KUKA KRL program: EPS_2_251112_SAMH04_A_20250918010312.src

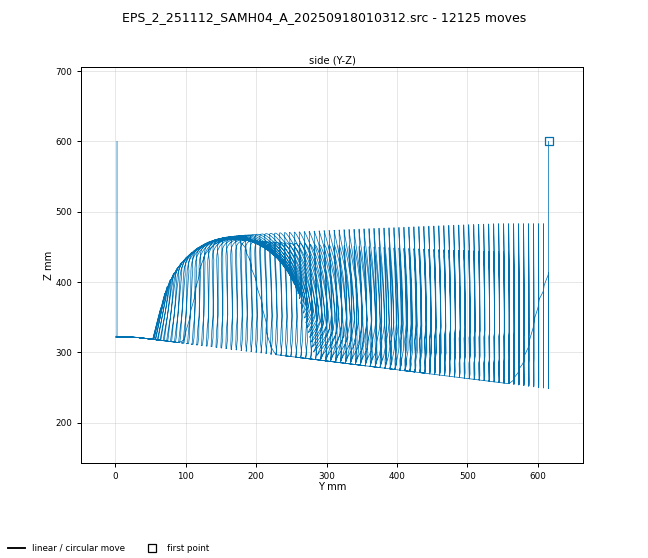
[picture p0: tool path of EPS_2_251112_SAMH04_A_20250918010312.src, 12125 of 12127 moves have a stored position in this frame; points joined in program order, loops and branches not executed]
&ACCESS RVP
&REL 4
&COMMENT QRS 19112012
&PARAM EDITMASK = *
DEF PART()
EXT BAS (BAS_COMMAND :IN,REAL :IN )
INT I
BAS (#INITMOV,0 )

;KUKA QRS Post kuka4.cps  Date:22-06-2017 !

File_ID=2832

QRS_PRE_INIT()

;Init var - Until changes are made in qrs_pre_init
Outlet_Square_prg=0
Inlet_1_Square_prg=0
Inlet_2_Square_prg=0
Inlet_3_Square_prg=0
Inlet_4_Square_prg=0
Inlet_5_Square_prg=0

Outlet_1={X 0.000, Y 541.230, Z 408.000, B 0.000, E1 0.000 }
Inlet_1={X 0.000, Y 544.070, Z 368.000, B 0.000, E1 90.000 }
Outlet_1_type=150
Inlet_1_type=150
;QRS#1=Sidecore dimensions
;QRS#2=150-6" PVC SDR 28
;QRS#3=150-6" PVC SDR 28
;QRS#4=
;QRS#5=
;QRS#6=
;QRS#7=
;QRS#8=
;QRS#9=10-06 PSX
;QRS#10=10-06 PSX
;QRS#11=
;QRS#12=
;QRS#13=
;QRS#14=
;QRS#15=
;QRS#16=1220x127x762 2,5'
;QRS#17=EPS Height
;QRS#18=483
;QRS#19=*
;QRS#20= UPDATED VERSION 22-06-2017
;QRS#21=*
Outlet_Square=070
Inlet_1_Square=070
Inlet_2_Square=0
Inlet_3_Square=0
Inlet_4_Square=0
Inlet_5_Square=0
Mill_Square=1
Outlet_Square_Prg=203
Inlet_1_Square_prg=203

QRS_INIT()

$ADVANCE=5

; T1
PTP {E1 173.474,E2 173.474}
PTP {X 0,Y 615.498,A -85,B 0,C 180,E1 173.474,E2 173.474,E3 0,E4 0,E5 0,E6 0}
QRS_SPEED_INIT()
LIN {X 0,Y 615.498,Z 600,A -85,B 0,C 180,E1 173.474,E2 173.474,E3 0,E4 0,E5 0,E6 0} C_VEL
LIN {X 0,Y 615.498,Z 427.975,A -85,B 0,C 180,E1 173.474,E2 173.474} C_VEL
LIN {X 0,Y 615.498,Z 415.28,A -85,B 0,C 180,E1 173.474,E2 173.474} C_VEL
LIN {X 0,Y 615.497,Z 413.833,A -85,B 0,C 180,E1 173.417,E2 173.417} C_VEL
LIN {X 0,Y 615.484,Z 405.601,A -85,B 0,C 180,E1 172.706,E2 172.706} C_VEL
LIN {X 0,Y 615.494,Z 395.743,A -85,B 0,C 180,E1 172.046,E2 172.046} C_VEL
LIN {X 0,Y 615.487,Z 388.006,A -85,B 0,C 180,E1 171.633,E2 171.633} C_VEL
LIN {X 0,Y 615.488,Z 379.171,A -85,B 0,C 180,E1 171.26,E2 171.26} C_VEL
LIN {X 0,Y 615.479,Z 369.995,A -85,B 0,C 180,E1 170.971,E2 170.971} C_VEL
LIN {X 0,Y 615.472,Z 360.409,A -85,B 0,C 180,E1 170.763,E2 170.763} C_VEL
LIN {X 0,Y 615.49,Z 301.527,A -85,B 0,C 180,E1 170.059,E2 170.059} C_VEL
LIN {X 0,Y 615.48,Z 284.33,A -85,B 0,C 180,E1 169.851,E2 169.851} C_VEL
LIN {X 0,Y 615.493,Z 270.832,A -85,B 0,C 180,E1 167.139,E2 167.139} C_VEL
LIN {X 0,Y 615.447,Z 257.533,A -85,B 0,C 180,E1 164.438,E2 164.438} C_VEL
LIN {X 0,Y 615.433,Z 248.511,A -85,B 0,C 180,E1 162.561,E2 162.561} C_VEL
LIN {X 0,Y 615.407,Z 248.511,A -85,B 0,C 180,E1 159.969,E2 159.969} C_VEL
LIN {X 0,Y 615.461,Z 248.512,A -85,B 0,C 180,E1 157.159,E2 157.159} C_VEL
LIN {X 0,Y 615.43,Z 248.511,A -85,B 0,C 180,E1 154.287,E2 154.287} C_VEL
LIN {X 0,Y 615.419,Z 248.511,A -85,B 0,C 180,E1 152.087,E2 152.087} C_VEL
LIN {X 0,Y 615.41,Z 248.511,A -85,B 0,C 180,E1 149.841,E2 149.841} C_VEL
LIN {X 0,Y 615.409,Z 248.511,A -85,B 0,C 180,E1 147.544,E2 147.544} C_VEL
LIN {X 0,Y 615.423,Z 248.512,A -85,B 0,C 180,E1 145.187,E2 145.187} C_VEL
LIN {X 0,Y 615.462,Z 248.512,A -85,B 0,C 180,E1 142.763,E2 142.763} C_VEL
LIN {X 0,Y 615.431,Z 248.511,A -85,B 0,C 180,E1 139.918,E2 139.918} C_VEL
LIN {X 0,Y 615.417,Z 248.51,A -85,B 0,C 180,E1 137.648,E2 137.648} C_VEL
LIN {X 0,Y 615.414,Z 248.511,A -85,B 0,C 180,E1 135.076,E2 135.076} C_VEL
LIN {X 0,Y 615.413,Z 248.511,A -85,B 0,C 180,E1 133.048,E2 133.048} C_VEL
LIN {X 0,Y 615.44,Z 248.512,A -85,B 0,C 180,E1 130.611,E2 130.611} C_VEL
LIN {X 0,Y 615.48,Z 248.512,A -85,B 0,C 180,E1 128.021,E2 128.021} C_VEL
LIN {X 0,Y 615.444,Z 248.51,A -85,B 0,C 180,E1 125.62,E2 125.62} C_VEL
LIN {X 0,Y 615.417,Z 248.51,A -85,B 0,C 180,E1 123.241,E2 123.241} C_VEL
LIN {X 0,Y 615.41,Z 248.511,A -85,B 0,C 180,E1 120.925,E2 120.925} C_VEL
LIN {X 0,Y 615.44,Z 248.51,A -85,B 0,C 180,E1 119.41,E2 119.41} C_VEL
LIN {X 0,Y 615.417,Z 248.51,A -85,B 0,C 180,E1 117.046,E2 117.046} C_VEL
LIN {X 0,Y 615.414,Z 248.511,A -85,B 0,C 180,E1 114.996,E2 114.996} C_VEL
LIN {X 0,Y 615.413,Z 248.51,A -85,B 0,C 180,E1 112.848,E2 112.848} C_VEL
LIN {X 0,Y 615.411,Z 248.511,A -85,B 0,C 180,E1 110.556,E2 110.556} C_VEL
LIN {X 0,Y 615.445,Z 248.512,A -85,B 0,C 180,E1 107.959,E2 107.959} C_VEL
LIN {X 0,Y 615.468,Z 248.509,A -85,B 0,C 180,E1 105.227,E2 105.227} C_VEL
LIN {X 0,Y 615.413,Z 248.51,A -85,B 0,C 180,E1 102.533,E2 102.533} C_VEL
LIN {X 0,Y 615.415,Z 248.51,A -85,B 0,C 180,E1 100.529,E2 100.529} C_VEL
LIN {X 0,Y 615.418,Z 248.51,A -85,B 0,C 180,E1 98.539,E2 98.539} C_VEL
LIN {X 0,Y 615.422,Z 248.51,A -85,B 0,C 180,E1 96.558,E2 96.558} C_VEL
LIN {X 0,Y 615.428,Z 248.509,A -85,B 0,C 180,E1 94.586,E2 94.586} C_VEL
LIN {X 0,Y 615.436,Z 248.509,A -85,B 0,C 180,E1 92.619,E2 92.619} C_VEL
LIN {X 0,Y 615.446,Z 248.509,A -85,B 0,C 180,E1 90.655,E2 90.655} C_VEL
LIN {X 0,Y 615.413,Z 248.51,A -85,B 0,C 180,E1 88.038,E2 88.038} C_VEL
LIN {X 0,Y 615.414,Z 248.51,A -85,B 0,C 180,E1 86.072,E2 86.072} C_VEL
LIN {X 0,Y 615.416,Z 248.51,A -85,B 0,C 180,E1 84.102,E2 84.102} C_VEL
LIN {X 0,Y 615.421,Z 248.509,A -85,B 0,C 180,E1 82.125,E2 82.125} C_VEL
LIN {X 0,Y 615.425,Z 248.509,A -85,B 0,C 180,E1 80.138,E2 80.138} C_VEL
LIN {X 0,Y 615.43,Z 248.509,A -85,B 0,C 180,E1 78.139,E2 78.139} C_VEL
LIN {X 0,Y 615.428,Z 248.509,A -85,B 0,C 180,E1 76.063,E2 76.063} C_VEL
LIN {X 0,Y 615.432,Z 248.51,A -85,B 0,C 180,E1 74.095,E2 74.095} C_VEL
LIN {X 0,Y 615.436,Z 248.509,A -85,B 0,C 180,E1 72.043,E2 72.043} C_VEL
LIN {X 0,Y 615.435,Z 248.509,A -85,B 0,C 180,E1 69.967,E2 69.967} C_VEL
LIN {X 0,Y 615.418,Z 248.509,A -85,B 0,C 180,E1 67.653,E2 67.653} C_VEL
LIN {X 0,Y 615.425,Z 248.509,A -85,B 0,C 180,E1 65.727,E2 65.727} C_VEL
LIN {X 0,Y 615.419,Z 248.509,A -85,B 0,C 180,E1 63.554,E2 63.554} C_VEL
LIN {X 0,Y 615.412,Z 248.51,A -85,B 0,C 180,E1 61.34,E2 61.34} C_VEL
LIN {X 0,Y 615.447,Z 248.509,A -85,B 0,C 180,E1 59.84,E2 59.84} C_VEL
LIN {X 0,Y 615.429,Z 248.509,A -85,B 0,C 180,E1 57.541,E2 57.541} C_VEL
LIN {X 0,Y 615.416,Z 248.509,A -85,B 0,C 180,E1 55.182,E2 55.182} C_VEL
LIN {X 0,Y 615.415,Z 248.51,A -85,B 0,C 180,E1 53.063,E2 53.063} C_VEL
LIN {X 0,Y 615.415,Z 248.51,A -85,B 0,C 180,E1 50.937,E2 50.937} C_VEL
LIN {X 0,Y 615.415,Z 248.51,A -85,B 0,C 180,E1 48.904,E2 48.904} C_VEL
LIN {X 0,Y 615.417,Z 248.51,A -85,B 0,C 180,E1 46.751,E2 46.751} C_VEL
LIN {X 0,Y 615.417,Z 248.509,A -85,B 0,C 180,E1 44.927,E2 44.927} C_VEL
LIN {X 0,Y 615.432,Z 248.511,A -85,B 0,C 180,E1 42.35,E2 42.35} C_VEL
LIN {X 0,Y 615.496,Z 248.513,A -85,B 0,C 180,E1 39.743,E2 39.743} C_VEL
LIN {X 0,Y 615.427,Z 248.508,A -85,B 0,C 180,E1 36.932,E2 36.932} C_VEL
LIN {X 0,Y 615.419,Z 248.509,A -85,B 0,C 180,E1 34.694,E2 34.694} C_VEL
LIN {X 0,Y 615.417,Z 248.509,A -85,B 0,C 180,E1 32.456,E2 32.456} C_VEL
LIN {X 0,Y 615.453,Z 248.512,A -85,B 0,C 180,E1 29.793,E2 29.793} C_VEL
LIN {X 0,Y 615.467,Z 248.507,A -85,B 0,C 180,E1 27.045,E2 27.045} C_VEL
LIN {X 0,Y 615.467,Z 248.507,A -85,B 0,C 180,E1 24.987,E2 24.987} C_VEL
LIN {X 0,Y 615.419,Z 248.509,A -85,B 0,C 180,E1 22.335,E2 22.335} C_VEL
LIN {X 0,Y 615.417,Z 248.51,A -85,B 0,C 180,E1 20.03,E2 20.03} C_VEL
LIN {X 0,Y 615.477,Z 248.513,A -85,B 0,C 180,E1 17.266,E2 17.266} C_VEL
LIN {X 0,Y 615.448,Z 248.507,A -85,B 0,C 180,E1 14.546,E2 14.546} C_VEL
LIN {X 0,Y 615.453,Z 248.507,A -85,B 0,C 180,E1 12.527,E2 12.527} C_VEL
LIN {X 0,Y 615.459,Z 248.507,A -85,B 0,C 180,E1 10.523,E2 10.523} C_VEL
LIN {X 0,Y 615.419,Z 248.509,A -85,B 0,C 180,E1 7.873,E2 7.873} C_VEL
LIN {X 0,Y 615.42,Z 248.508,A -85,B 0,C 180,E1 5.896,E2 5.896} C_VEL
LIN {X 0,Y 615.424,Z 248.508,A -85,B 0,C 180,E1 3.925,E2 3.925} C_VEL
LIN {X 0,Y 615.428,Z 248.508,A -85,B 0,C 180,E1 1.96,E2 1.96} C_VEL
LIN {X 0,Y 615.435,Z 248.507,A -85,B 0,C 180,E1 -0.003,E2 -0.003} C_VEL
LIN {X 0,Y 615.443,Z 248.507,A -85,B 0,C 180,E1 -1.966,E2 -1.966} C_VEL
LIN {X 0,Y 615.453,Z 248.506,A -85,B 0,C 180,E1 -3.932,E2 -3.932} C_VEL
LIN {X 0,Y 615.419,Z 248.509,A -85,B 0,C 180,E1 -6.56,E2 -6.56} C_VEL
LIN {X 0,Y 615.42,Z 248.508,A -85,B 0,C 180,E1 -8.54,E2 -8.54} C_VEL
LIN {X 0,Y 615.422,Z 248.509,A -85,B 0,C 180,E1 -10.866,E2 -10.866} C_VEL
LIN {X 0,Y 615.438,Z 248.511,A -85,B 0,C 180,E1 -13.205,E2 -13.205} C_VEL
LIN {X 0,Y 615.488,Z 248.509,A -85,B 0,C 180,E1 -15.908,E2 -15.908} C_VEL
LIN {X 0,Y 615.427,Z 248.507,A -85,B 0,C 180,E1 -18.65,E2 -18.65} C_VEL
LIN {X 0,Y 615.426,Z 248.507,A -85,B 0,C 180,E1 -20.735,E2 -20.735} C_VEL
LIN {X 0,Y 615.422,Z 248.508,A -85,B 0,C 180,E1 -22.849,E2 -22.849} C_VEL
LIN {X 0,Y 615.421,Z 248.508,A -85,B 0,C 180,E1 -24.997,E2 -24.997} C_VEL
LIN {X 0,Y 615.419,Z 248.509,A -85,B 0,C 180,E1 -27.182,E2 -27.182} C_VEL
LIN {X 0,Y 615.453,Z 248.511,A -85,B 0,C 180,E1 -29.793,E2 -29.793} C_VEL
LIN {X 0,Y 615.491,Z 248.504,A -85,B 0,C 180,E1 -32.459,E2 -32.459} C_VEL
LIN {X 0,Y 615.447,Z 248.507,A -85,B 0,C 180,E1 -34.819,E2 -34.819} C_VEL
LIN {X 0,Y 615.425,Z 248.507,A -85,B 0,C 180,E1 -37.248,E2 -37.248} C_VEL
LIN {X 0,Y 615.454,Z 248.511,A -85,B 0,C 180,E1 -40.088,E2 -40.088} C_VEL
LIN {X 0,Y 615.45,Z 248.506,A -85,B 0,C 180,E1 -43.046,E2 -43.046} C_VEL
LIN {X 0,Y 615.425,Z 248.509,A -85,B 0,C 180,E1 -45.847,E2 -45.847} C_VEL
LIN {X 0,Y 615.426,Z 248.509,A -85,B 0,C 180,E1 -47.927,E2 -47.927} C_VEL
LIN {X 0,Y 615.444,Z 248.51,A -85,B 0,C 180,E1 -50.249,E2 -50.249} C_VEL
LIN {X 0,Y 615.484,Z 248.504,A -85,B 0,C 180,E1 -53.065,E2 -53.065} C_VEL
LIN {X 0,Y 615.423,Z 248.508,A -85,B 0,C 180,E1 -55.976,E2 -55.976} C_VEL
LIN {X 0,Y 615.486,Z 248.516,A -85,B 0,C 180,E1 -58.915,E2 -58.915} C_VEL
LIN {X 0,Y 615.452,Z 248.505,A -85,B 0,C 180,E1 -61.557,E2 -61.557} C_VEL
LIN {X 0,Y 615.458,Z 248.505,A -85,B 0,C 180,E1 -63.556,E2 -63.556} C_VEL
LIN {X 0,Y 615.428,Z 248.507,A -85,B 0,C 180,E1 -66.005,E2 -66.005} C_VEL
LIN {X 0,Y 615.422,Z 248.509,A -85,B 0,C 180,E1 -68.391,E2 -68.391} C_VEL
LIN {X 0,Y 615.429,Z 248.57,A -85,B 0,C 180,E1 -68.567,E2 -68.567} C_VEL
LIN {X 0,Y 615.488,Z 265.289,A -85,B 0,C 180,E1 -71.183,E2 -71.183} C_VEL
LIN {X 0,Y 615.496,Z 282.488,A -85,B 0,C 180,E1 -73.833,E2 -73.833} C_VEL
LIN {X 0,Y 615.445,Z 300.903,A -85,B 0,C 180,E1 -76.631,E2 -76.631} C_VEL
LIN {X 0,Y 615.481,Z 318.596,A -85,B 0,C 180,E1 -79.295,E2 -79.295} C_VEL
LIN {X 0,Y 615.492,Z 322.424,A -85,B 0,C 180,E1 -79.869,E2 -79.869} C_VEL
LIN {X 0,Y 615.465,Z 400.026,A -85,B 0,C 180,E1 -80.802,E2 -80.802} C_VEL
LIN {X 0,Y 615.457,Z 409.755,A -85,B 0,C 180,E1 -81.009,E2 -81.009} C_VEL
LIN {X 0,Y 615.463,Z 420.197,A -85,B 0,C 180,E1 -81.34,E2 -81.34} C_VEL
LIN {X 0,Y 615.491,Z 430.45,A -85,B 0,C 180,E1 -81.795,E2 -81.795} C_VEL
LIN {X 0,Y 615.478,Z 440.219,A -85,B 0,C 180,E1 -82.373,E2 -82.373} C_VEL
LIN {X 0,Y 615.493,Z 447.948,A -85,B 0,C 180,E1 -82.943,E2 -82.943} C_VEL
LIN {X 0,Y 615.498,Z 455.346,A -85,B 0,C 180,E1 -83.609,E2 -83.609} C_VEL
LIN {X 0,Y 615.498,Z 462.747,A -85,B 0,C 180,E1 -84.432,E2 -84.432} C_VEL
LIN {X 0,Y 615.497,Z 468.54,A -85,B 0,C 180,E1 -85.253,E2 -85.253} C_VEL
LIN {X 0,Y 615.495,Z 473.105,A -85,B 0,C 180,E1 -86.073,E2 -86.073} C_VEL
LIN {X 0,Y 615.493,Z 476.073,A -85,B 0,C 180,E1 -86.728,E2 -86.728} C_VEL
LIN {X 0,Y 615.494,Z 478.36,A -85,B 0,C 180,E1 -87.383,E2 -87.383} C_VEL
LIN {X 0,Y 615.499,Z 480.088,A -85,B 0,C 180,E1 -88.038,E2 -88.038} C_VEL
LIN {X 0,Y 615.493,Z 481.331,A -85,B 0,C 180,E1 -88.693,E2 -88.693} C_VEL
LIN {X 0,Y 615.492,Z 482.105,A -85,B 0,C 180,E1 -89.347,E2 -89.347} C_VEL
LIN {X 0,Y 615.491,Z 482.389,A -85,B 0,C 180,E1 -90.001,E2 -90.001} C_VEL
LIN {X 0,Y 615.491,Z 482.104,A -85,B 0,C 180,E1 -90.655,E2 -90.655} C_VEL
LIN {X 0,Y 615.493,Z 481.328,A -85,B 0,C 180,E1 -91.31,E2 -91.31} C_VEL
LIN {X 0,Y 615.499,Z 480.082,A -85,B 0,C 180,E1 -91.964,E2 -91.964} C_VEL
LIN {X 0,Y 615.488,Z 477.217,A -85,B 0,C 180,E1 -92.946,E2 -92.946} C_VEL
LIN {X 0,Y 615.493,Z 474.598,A -85,B 0,C 180,E1 -93.602,E2 -93.602} C_VEL
LIN {X 0,Y 615.495,Z 469.476,A -85,B 0,C 180,E1 -94.586,E2 -94.586} C_VEL
LIN {X 0,Y 615.495,Z 463.961,A -85,B 0,C 180,E1 -95.406,E2 -95.406} C_VEL
LIN {X 0,Y 615.499,Z 457.008,A -85,B 0,C 180,E1 -96.228,E2 -96.228} C_VEL
LIN {X 0,Y 615.495,Z 449.857,A -85,B 0,C 180,E1 -96.901,E2 -96.901} C_VEL
LIN {X 0,Y 615.477,Z 442.609,A -85,B 0,C 180,E1 -97.464,E2 -97.464} C_VEL
LIN {X 0,Y 615.495,Z 434.851,A -85,B 0,C 180,E1 -97.959,E2 -97.959} C_VEL
LIN {X 0,Y 615.484,Z 426.894,A -85,B 0,C 180,E1 -98.372,E2 -98.372} C_VEL
LIN {X 0,Y 615.459,Z 417.736,A -85,B 0,C 180,E1 -98.745,E2 -98.745} C_VEL
LIN {X 0,Y 615.457,Z 409.665,A -85,B 0,C 180,E1 -98.993,E2 -98.993} C_VEL
LIN {X 0,Y 615.465,Z 399.886,A -85,B 0,C 180,E1 -99.2,E2 -99.2} C_VEL
LIN {X 0,Y 615.492,Z 322.409,A -85,B 0,C 180,E1 -100.133,E2 -100.133} C_VEL
LIN {X 0,Y 615.47,Z 303.108,A -85,B 0,C 180,E1 -103.035,E2 -103.035} C_VEL
LIN {X 0,Y 615.462,Z 285.317,A -85,B 0,C 180,E1 -105.737,E2 -105.737} C_VEL
LIN {X 0,Y 615.495,Z 266.648,A -85,B 0,C 180,E1 -108.606,E2 -108.606} C_VEL
LIN {X 0,Y 615.441,Z 249.669,A -85,B 0,C 180,E1 -111.259,E2 -111.259} C_VEL
LIN {X 0,Y 615.427,Z 248.51,A -85,B 0,C 180,E1 -111.479,E2 -111.479} C_VEL
LIN {X 0,Y 615.423,Z 248.51,A -85,B 0,C 180,E1 -113.56,E2 -113.56} C_VEL
LIN {X 0,Y 615.417,Z 248.51,A -85,B 0,C 180,E1 -115.72,E2 -115.72} C_VEL
LIN {X 0,Y 615.413,Z 248.511,A -85,B 0,C 180,E1 -117.92,E2 -117.92} C_VEL
LIN {X 0,Y 615.415,Z 248.512,A -85,B 0,C 180,E1 -120.165,E2 -120.165} C_VEL
LIN {X 0,Y 615.436,Z 248.513,A -85,B 0,C 180,E1 -122.461,E2 -122.461} C_VEL
LIN {X 0,Y 615.481,Z 248.513,A -85,B 0,C 180,E1 -124.816,E2 -124.816} C_VEL
LIN {X 0,Y 615.466,Z 248.509,A -85,B 0,C 180,E1 -127.244,E2 -127.244} C_VEL
LIN {X 0,Y 615.426,Z 248.509,A -85,B 0,C 180,E1 -129.756,E2 -129.756} C_VEL
LIN {X 0,Y 615.423,Z 248.509,A -85,B 0,C 180,E1 -132.072,E2 -132.072} C_VEL
LIN {X 0,Y 615.427,Z 248.508,A -85,B 0,C 180,E1 -134.156,E2 -134.156} C_VEL
LIN {X 0,Y 615.431,Z 248.507,A -85,B 0,C 180,E1 -136.009,E2 -136.009} C_VEL
LIN {X 0,Y 615.444,Z 248.51,A -85,B 0,C 180,E1 -138.521,E2 -138.521} C_VEL
LIN {X 0,Y 615.498,Z 248.51,A -85,B 0,C 180,E1 -141.095,E2 -141.095} C_VEL
LIN {X 0,Y 615.478,Z 248.501,A -85,B 0,C 180,E1 -143.573,E2 -143.573} C_VEL
LIN {X 0,Y 615.456,Z 248.501,A -85,B 0,C 180,E1 -145.974,E2 -145.974} C_VEL
LIN {X 0,Y 615.449,Z 248.504,A -85,B 0,C 180,E1 -148.311,E2 -148.311} C_VEL
LIN {X 0,Y 615.457,Z 248.506,A -85,B 0,C 180,E1 -150.59,E2 -150.59} C_VEL
LIN {X 0,Y 615.483,Z 248.511,A -85,B 0,C 180,E1 -152.957,E2 -152.957} C_VEL
LIN {X 0,Y 615.483,Z 248.495,A -85,B 0,C 180,E1 -155.994,E2 -155.994} C_VEL
LIN {X 0,Y 615.463,Z 248.503,A -85,B 0,C 180,E1 -158.565,E2 -158.565} C_VEL
LIN {X 0,Y 615.484,Z 248.509,A -85,B 0,C 180,E1 -161.352,E2 -161.352} C_VEL
LIN {X 0,Y 615.469,Z 248.532,A -85,B 0,C 180,E1 -162.684,E2 -162.684} C_VEL
LIN {X 0,Y 615.469,Z 262.046,A -85,B 0,C 180,E1 -165.448,E2 -165.448} C_VEL
LIN {X 0,Y 615.486,Z 275.335,A -85,B 0,C 180,E1 -168.136,E2 -168.136} C_VEL
LIN {X 0,Y 615.463,Z 284.368,A -85,B 0,C 180,E1 -169.948,E2 -169.948} C_VEL
LIN {X 0,Y 615.437,Z 359.563,A -85,B 0,C 180,E1 -170.839,E2 -170.839} C_VEL
LIN {X 0,Y 615.429,Z 367.804,A -85,B 0,C 180,E1 -171.005,E2 -171.005} C_VEL
LIN {X 0,Y 615.427,Z 376.389,A -85,B 0,C 180,E1 -171.253,E2 -171.253} C_VEL
LIN {X 0,Y 615.44,Z 384.013,A -85,B 0,C 180,E1 -171.543,E2 -171.543} C_VEL
LIN {X 0,Y 615.485,Z 392.534,A -85,B 0,C 180,E1 -171.956,E2 -171.956} C_VEL
LIN {X 0,Y 615.491,Z 400.706,A -85,B 0,C 180,E1 -172.452,E2 -172.452} C_VEL
LIN {X 0,Y 615.492,Z 407.367,A -85,B 0,C 180,E1 -172.94,E2 -172.94} C_VEL
LIN {X 0,Y 615.498,Z 413.154,A -85,B 0,C 180,E1 -173.441,E2 -173.441} C_VEL
LIN {X 0,Y 615.499,Z 419.509,A -85,B 0,C 180,E1 -174.099,E2 -174.099} C_VEL
LIN {X 0,Y 615.495,Z 425.963,A -85,B 0,C 180,E1 -174.92,E2 -174.92} C_VEL
LIN {X 0,Y 615.492,Z 431.105,A -85,B 0,C 180,E1 -175.741,E2 -175.741} C_VEL
LIN {X 0,Y 615.493,Z 435.874,A -85,B 0,C 180,E1 -176.724,E2 -176.724} C_VEL
LIN {X 0,Y 615.493,Z 438.189,A -85,B 0,C 180,E1 -177.379,E2 -177.379} C_VEL
LIN {X 0,Y 615.494,Z 439.969,A -85,B 0,C 180,E1 -178.034,E2 -178.034} C_VEL
LIN {X 0,Y 615.496,Z 441.261,A -85,B 0,C 180,E1 -178.688,E2 -178.688} C_VEL
LIN {X 0,Y 615.491,Z 442.082,A -85,B 0,C 180,E1 -179.343,E2 -179.343} C_VEL
LIN {X 0,Y 615.492,Z 442.384,A -85,B 0,C 180,E1 -179.997,E2 -179.997} C_VEL
LIN {X 0,Y 615.494,Z 442.126,A -85,B 0,C 180,E1 -180.651,E2 -180.651} C_VEL
LIN {X 0,Y 615.494,Z 441.398,A -85,B 0,C 180,E1 -181.305,E2 -181.305} C_VEL
LIN {X 0,Y 615.498,Z 440.203,A -85,B 0,C 180,E1 -181.96,E2 -181.96} C_VEL
LIN {X 0,Y 615.491,Z 437.388,A -85,B 0,C 180,E1 -182.942,E2 -182.942} C_VEL
LIN {X 0,Y 615.491,Z 434.826,A -85,B 0,C 180,E1 -183.597,E2 -183.597} C_VEL
LIN {X 0,Y 615.498,Z 429.763,A -85,B 0,C 180,E1 -184.581,E2 -184.581} C_VEL
LIN {X 0,Y 615.496,Z 424.313,A -85,B 0,C 180,E1 -185.402,E2 -185.402} C_VEL
LIN {X 0,Y 615.497,Z 417.487,A -85,B 0,C 180,E1 -186.224,E2 -186.224} C_VEL
LIN {X 0,Y 615.497,Z 413.833,A -85,B 0,C 180,E1 -186.583,E2 -186.583} C_VEL
LIN {X 0,Y 614.837,Z 409.751,A -85,B 0,C 180,E1 -186.976,E2 -186.976} C_VEL
LIN {X 0,Y 611.99,Z 402.713,A -85,B 0,C 180,E1 -187.58,E2 -187.58} C_VEL
LIN {X 0,Y 609.145,Z 395.09,A -85,B 0,C 180,E1 -188.111,E2 -188.111} C_VEL
LIN {X 0,Y 608.48,Z 390,A -85,B 0,C 180,E1 -188.385,E2 -188.385} C_VEL
LIN {X 0,Y 608.479,Z 379.497,A -85,B 0,C 180,E1 -188.841,E2 -188.841} C_VEL
LIN {X 0,Y 608.494,Z 369.524,A -85,B 0,C 180,E1 -189.155,E2 -189.155} C_VEL
LIN {X 0,Y 608.501,Z 360.878,A -85,B 0,C 180,E1 -189.343,E2 -189.343} C_VEL
LIN {X 0,Y 608.5,Z 328.822,A -85,B 0,C 180,E1 -189.742,E2 -189.742} C_VEL
LIN {X 0,Y 608.437,Z 284.646,A -85,B 0,C 180,E1 -190.268,E2 -190.268} C_VEL
LIN {X 0,Y 608.46,Z 271.068,A -85,B 0,C 180,E1 -193.012,E2 -193.012} C_VEL
LIN {X 0,Y 608.413,Z 257.699,A -85,B 0,C 180,E1 -195.747,E2 -195.747} C_VEL
LIN {X 0,Y 608.408,Z 249.507,A -85,B 0,C 180,E1 -197.473,E2 -197.473} C_VEL
LIN {X 0,Y 608.406,Z 249.507,A -85,B 0,C 180,E1 -199.567,E2 -199.567} C_VEL
LIN {X 0,Y 608.418,Z 249.505,A -85,B 0,C 180,E1 -201.689,E2 -201.689} C_VEL
LIN {X 0,Y 608.41,Z 249.507,A -85,B 0,C 180,E1 -204.568,E2 -204.568} C_VEL
LIN {X 0,Y 608.467,Z 249.509,A -85,B 0,C 180,E1 -207.204,E2 -207.204} C_VEL
LIN {X 0,Y 608.394,Z 249.507,A -85,B 0,C 180,E1 -209.959,E2 -209.959} C_VEL
LIN {X 0,Y 608.393,Z 249.507,A -85,B 0,C 180,E1 -212.511,E2 -212.511} C_VEL
LIN {X 0,Y 608.394,Z 249.509,A -85,B 0,C 180,E1 -214.897,E2 -214.897} C_VEL
LIN {X 0,Y 608.428,Z 249.509,A -85,B 0,C 180,E1 -217.742,E2 -217.742} C_VEL
LIN {X 0,Y 608.399,Z 249.506,A -85,B 0,C 180,E1 -220.322,E2 -220.322} C_VEL
LIN {X 0,Y 608.387,Z 249.508,A -85,B 0,C 180,E1 -222.958,E2 -222.958} C_VEL
LIN {X 0,Y 608.445,Z 249.511,A -85,B 0,C 180,E1 -225.729,E2 -225.729} C_VEL
LIN {X 0,Y 608.462,Z 249.506,A -85,B 0,C 180,E1 -227.938,E2 -227.938} C_VEL
LIN {X 0,Y 608.382,Z 249.508,A -85,B 0,C 180,E1 -230.703,E2 -230.703} C_VEL
LIN {X 0,Y 608.383,Z 249.508,A -85,B 0,C 180,E1 -233.079,E2 -233.079} C_VEL
LIN {X 0,Y 608.424,Z 249.506,A -85,B 0,C 180,E1 -235.527,E2 -235.527} C_VEL
LIN {X 0,Y 608.432,Z 249.511,A -85,B 0,C 180,E1 -237.903,E2 -237.903} C_VEL
LIN {X 0,Y 608.475,Z 249.505,A -85,B 0,C 180,E1 -240.22,E2 -240.22} C_VEL
LIN {X 0,Y 608.382,Z 249.508,A -85,B 0,C 180,E1 -243.222,E2 -243.222} C_VEL
LIN {X 0,Y 608.409,Z 249.507,A -85,B 0,C 180,E1 -244.696,E2 -244.696} C_VEL
LIN {X 0,Y 608.403,Z 249.507,A -85,B 0,C 180,E1 -246.873,E2 -246.873} C_VEL
LIN {X 0,Y 608.396,Z 249.506,A -85,B 0,C 180,E1 -249.321,E2 -249.321} C_VEL
LIN {X 0,Y 608.396,Z 249.508,A -85,B 0,C 180,E1 -251.826,E2 -251.826} C_VEL
LIN {X 0,Y 608.443,Z 249.51,A -85,B 0,C 180,E1 -254.592,E2 -254.592} C_VEL
LIN {X 0,Y 608.416,Z 249.504,A -85,B 0,C 180,E1 -257.321,E2 -257.321} C_VEL
LIN {X 0,Y 608.402,Z 249.506,A -85,B 0,C 180,E1 -259.348,E2 -259.348} C_VEL
LIN {X 0,Y 608.399,Z 249.507,A -85,B 0,C 180,E1 -261.362,E2 -261.362} C_VEL
LIN {X 0,Y 608.412,Z 249.505,A -85,B 0,C 180,E1 -263.366,E2 -263.366} C_VEL
LIN {X 0,Y 608.402,Z 249.507,A -85,B 0,C 180,E1 -265.361,E2 -265.361} C_VEL
LIN {X 0,Y 608.428,Z 249.505,A -85,B 0,C 180,E1 -267.351,E2 -267.351} C_VEL
LIN {X 0,Y 608.404,Z 249.505,A -85,B 0,C 180,E1 -269.999,E2 -269.999} C_VEL
LIN {X 0,Y 608.438,Z 249.506,A -85,B 0,C 180,E1 -272.647,E2 -272.647} C_VEL
LIN {X 0,Y 608.448,Z 249.506,A -85,B 0,C 180,E1 -275.301,E2 -275.301} C_VEL
LIN {X 0,Y 608.413,Z 249.504,A -85,B 0,C 180,E1 -277.967,E2 -277.967} C_VEL
LIN {X 0,Y 608.393,Z 249.507,A -85,B 0,C 180,E1 -279.977,E2 -279.977} C_VEL
LIN {X 0,Y 608.402,Z 249.506,A -85,B 0,C 180,E1 -282,E2 -282} C_VEL
LIN {X 0,Y 608.402,Z 249.506,A -85,B 0,C 180,E1 -284.038,E2 -284.038} C_VEL
LIN {X 0,Y 608.4,Z 249.506,A -85,B 0,C 180,E1 -286.53,E2 -286.53} C_VEL
LIN {X 0,Y 608.401,Z 249.508,A -85,B 0,C 180,E1 -288.87,E2 -288.87} C_VEL
LIN {X 0,Y 608.448,Z 249.507,A -85,B 0,C 180,E1 -291.691,E2 -291.691} C_VEL
LIN {X 0,Y 608.393,Z 249.506,A -85,B 0,C 180,E1 -294.572,E2 -294.572} C_VEL
LIN {X 0,Y 608.386,Z 249.507,A -85,B 0,C 180,E1 -296.776,E2 -296.776} C_VEL
LIN {X 0,Y 608.477,Z 249.506,A -85,B 0,C 180,E1 -299.777,E2 -299.777} C_VEL
LIN {X 0,Y 608.403,Z 249.506,A -85,B 0,C 180,E1 -302.525,E2 -302.525} C_VEL
LIN {X 0,Y 608.411,Z 249.504,A -85,B 0,C 180,E1 -304.911,E2 -304.911} C_VEL
LIN {X 0,Y 608.441,Z 249.509,A -85,B 0,C 180,E1 -307.746,E2 -307.746} C_VEL
LIN {X 0,Y 608.457,Z 249.503,A -85,B 0,C 180,E1 -310.339,E2 -310.339} C_VEL
LIN {X 0,Y 608.444,Z 249.506,A -85,B 0,C 180,E1 -312.341,E2 -312.341} C_VEL
LIN {X 0,Y 608.4,Z 249.506,A -85,B 0,C 180,E1 -314.799,E2 -314.799} C_VEL
LIN {X 0,Y 608.391,Z 249.507,A -85,B 0,C 180,E1 -317.042,E2 -317.042} C_VEL
LIN {X 0,Y 608.401,Z 249.508,A -85,B 0,C 180,E1 -319.7,E2 -319.7} C_VEL
LIN {X 0,Y 608.436,Z 249.512,A -85,B 0,C 180,E1 -322.258,E2 -322.258} C_VEL
LIN {X 0,Y 608.422,Z 249.504,A -85,B 0,C 180,E1 -325.095,E2 -325.095} C_VEL
LIN {X 0,Y 608.397,Z 249.506,A -85,B 0,C 180,E1 -327.484,E2 -327.484} C_VEL
LIN {X 0,Y 608.437,Z 249.507,A -85,B 0,C 180,E1 -330.225,E2 -330.225} C_VEL
LIN {X 0,Y 608.408,Z 249.506,A -85,B 0,C 180,E1 -333.229,E2 -333.229} C_VEL
LIN {X 0,Y 608.394,Z 249.507,A -85,B 0,C 180,E1 -335.861,E2 -335.861} C_VEL
LIN {X 0,Y 608.433,Z 249.505,A -85,B 0,C 180,E1 -338.312,E2 -338.312} C_VEL
LIN {X 0,Y 608.433,Z 249.505,A -85,B 0,C 180,E1 -341.289,E2 -341.289} C_VEL
LIN {X 0,Y 608.4,Z 249.505,A -85,B 0,C 180,E1 -343.909,E2 -343.909} C_VEL
LIN {X 0,Y 608.4,Z 249.505,A -85,B 0,C 180,E1 -346.001,E2 -346.001} C_VEL
LIN {X 0,Y 608.449,Z 249.505,A -85,B 0,C 180,E1 -348.68,E2 -348.68} C_VEL
LIN {X 0,Y 608.436,Z 249.507,A -85,B 0,C 180,E1 -351.368,E2 -351.368} C_VEL
LIN {X 0,Y 608.402,Z 249.505,A -85,B 0,C 180,E1 -354.036,E2 -354.036} C_VEL
LIN {X 0,Y 608.397,Z 249.506,A -85,B 0,C 180,E1 -356.029,E2 -356.029} C_VEL
LIN {X 0,Y 608.402,Z 249.506,A -85,B 0,C 180,E1 -358.017,E2 -358.017} C_VEL
LIN {X 0,Y 608.429,Z 249.503,A -85,B 0,C 180,E1 -360.003,E2 -360.003} C_VEL
LIN {X 0,Y 608.413,Z 249.506,A -85,B 0,C 180,E1 -361.989,E2 -361.989} C_VEL
LIN {X 0,Y 608.419,Z 249.505,A -85,B 0,C 180,E1 -363.977,E2 -363.977} C_VEL
LIN {X 0,Y 608.417,Z 249.504,A -85,B 0,C 180,E1 -366.636,E2 -366.636} C_VEL
LIN {X 0,Y 608.44,Z 249.507,A -85,B 0,C 180,E1 -369.309,E2 -369.309} C_VEL
LIN {X 0,Y 608.446,Z 249.505,A -85,B 0,C 180,E1 -372.003,E2 -372.003} C_VEL
LIN {X 0,Y 608.392,Z 249.506,A -85,B 0,C 180,E1 -374.725,E2 -374.725} C_VEL
LIN {X 0,Y 608.402,Z 249.505,A -85,B 0,C 180,E1 -376.788,E2 -376.788} C_VEL
LIN {X 0,Y 608.417,Z 249.503,A -85,B 0,C 180,E1 -378.873,E2 -378.873} C_VEL
LIN {X 0,Y 608.444,Z 249.508,A -85,B 0,C 180,E1 -381.695,E2 -381.695} C_VEL
LIN {X 0,Y 608.425,Z 249.504,A -85,B 0,C 180,E1 -384.574,E2 -384.574} C_VEL
LIN {X 0,Y 608.403,Z 249.505,A -85,B 0,C 180,E1 -387.197,E2 -387.197} C_VEL
LIN {X 0,Y 608.471,Z 249.505,A -85,B 0,C 180,E1 -389.976,E2 -389.976} C_VEL
LIN {X 0,Y 608.427,Z 249.503,A -85,B 0,C 180,E1 -392.883,E2 -392.883} C_VEL
LIN {X 0,Y 608.397,Z 249.506,A -85,B 0,C 180,E1 -395.282,E2 -395.282} C_VEL
LIN {X 0,Y 608.443,Z 249.51,A -85,B 0,C 180,E1 -398.24,E2 -398.24} C_VEL
LIN {X 0,Y 608.406,Z 249.506,A -85,B 0,C 180,E1 -401.182,E2 -401.182} C_VEL
LIN {X 0,Y 608.426,Z 249.503,A -85,B 0,C 180,E1 -403.307,E2 -403.307} C_VEL
LIN {X 0,Y 608.431,Z 249.506,A -85,B 0,C 180,E1 -406.129,E2 -406.129} C_VEL
LIN {X 0,Y 608.451,Z 249.507,A -85,B 0,C 180,E1 -408.825,E2 -408.825} C_VEL
LIN {X 0,Y 608.42,Z 249.503,A -85,B 0,C 180,E1 -411.767,E2 -411.767} C_VEL
LIN {X 0,Y 608.402,Z 249.506,A -85,B 0,C 180,E1 -413.961,E2 -413.961} C_VEL
LIN {X 0,Y 608.422,Z 249.506,A -85,B 0,C 180,E1 -416.329,E2 -416.329} C_VEL
LIN {X 0,Y 608.441,Z 249.509,A -85,B 0,C 180,E1 -418.734,E2 -418.734} C_VEL
LIN {X 0,Y 608.408,Z 249.505,A -85,B 0,C 180,E1 -421.733,E2 -421.733} C_VEL
LIN {X 0,Y 608.423,Z 249.503,A -85,B 0,C 180,E1 -424.289,E2 -424.289} C_VEL
LIN {X 0,Y 608.43,Z 249.509,A -85,B 0,C 180,E1 -426.877,E2 -426.877} C_VEL
LIN {X 0,Y 608.443,Z 249.699,A -85,B 0,C 180,E1 -428.487,E2 -428.487} C_VEL
LIN {X 0,Y 608.507,Z 265.33,A -85,B 0,C 180,E1 -430.959,E2 -430.959} C_VEL
LIN {X 0,Y 608.509,Z 283.239,A -85,B 0,C 180,E1 -433.743,E2 -433.743} C_VEL
LIN {X 0,Y 608.433,Z 302.177,A -85,B 0,C 180,E1 -436.644,E2 -436.644} C_VEL
LIN {X 0,Y 608.44,Z 319.064,A -85,B 0,C 180,E1 -439.204,E2 -439.204} C_VEL
LIN {X 0,Y 608.473,Z 322.694,A -85,B 0,C 180,E1 -439.751,E2 -439.751} C_VEL
LIN {X 0,Y 608.489,Z 400.522,A -85,B 0,C 180,E1 -440.696,E2 -440.696} C_VEL
LIN {X 0,Y 608.47,Z 410.955,A -85,B 0,C 180,E1 -440.926,E2 -440.926} C_VEL
LIN {X 0,Y 608.471,Z 421.648,A -85,B 0,C 180,E1 -441.282,E2 -441.282} C_VEL
LIN {X 0,Y 608.473,Z 432.255,A -85,B 0,C 180,E1 -441.784,E2 -441.784} C_VEL
LIN {X 0,Y 608.458,Z 440.56,A -85,B 0,C 180,E1 -442.285,E2 -442.285} C_VEL
LIN {X 0,Y 608.459,Z 448.416,A -85,B 0,C 180,E1 -442.869,E2 -442.869} C_VEL
LIN {X 0,Y 608.466,Z 455.367,A -85,B 0,C 180,E1 -443.497,E2 -443.497} C_VEL
LIN {X 0,Y 608.469,Z 463.201,A -85,B 0,C 180,E1 -444.367,E2 -444.367} C_VEL
LIN {X 0,Y 608.448,Z 469.034,A -85,B 0,C 180,E1 -445.197,E2 -445.197} C_VEL
LIN {X 0,Y 608.433,Z 473.636,A -85,B 0,C 180,E1 -446.027,E2 -446.027} C_VEL
LIN {X 0,Y 608.425,Z 476.626,A -85,B 0,C 180,E1 -446.69,E2 -446.69} C_VEL
LIN {X 0,Y 608.423,Z 478.935,A -85,B 0,C 180,E1 -447.353,E2 -447.353} C_VEL
LIN {X 0,Y 608.444,Z 480.681,A -85,B 0,C 180,E1 -448.015,E2 -448.015} C_VEL
LIN {X 0,Y 608.446,Z 481.935,A -85,B 0,C 180,E1 -448.677,E2 -448.677} C_VEL
LIN {X 0,Y 608.434,Z 482.714,A -85,B 0,C 180,E1 -449.339,E2 -449.339} C_VEL
LIN {X 0,Y 608.431,Z 483,A -85,B 0,C 180,E1 -450.001,E2 -450.001} C_VEL
LIN {X 0,Y 608.434,Z 482.713,A -85,B 0,C 180,E1 -450.663,E2 -450.663} C_VEL
LIN {X 0,Y 608.446,Z 481.932,A -85,B 0,C 180,E1 -451.325,E2 -451.325} C_VEL
LIN {X 0,Y 608.444,Z 480.675,A -85,B 0,C 180,E1 -451.987,E2 -451.987} C_VEL
LIN {X 0,Y 608.444,Z 477.782,A -85,B 0,C 180,E1 -452.981,E2 -452.981} C_VEL
LIN {X 0,Y 608.446,Z 475.141,A -85,B 0,C 180,E1 -453.643,E2 -453.643} C_VEL
LIN {X 0,Y 608.431,Z 469.979,A -85,B 0,C 180,E1 -454.639,E2 -454.639} C_VEL
LIN {X 0,Y 608.46,Z 464.422,A -85,B 0,C 180,E1 -455.469,E2 -455.469} C_VEL
LIN {X 0,Y 608.456,Z 456.677,A -85,B 0,C 180,E1 -456.375,E2 -456.375} C_VEL
LIN {X 0,Y 608.453,Z 449.402,A -85,B 0,C 180,E1 -457.05,E2 -457.05} C_VEL
LIN {X 0,Y 608.459,Z 441.745,A -85,B 0,C 180,E1 -457.634,E2 -457.634} C_VEL
LIN {X 0,Y 608.493,Z 433.701,A -85,B 0,C 180,E1 -458.135,E2 -458.135} C_VEL
LIN {X 0,Y 608.475,Z 425.366,A -85,B 0,C 180,E1 -458.553,E2 -458.553} C_VEL
LIN {X 0,Y 608.452,Z 416.859,A -85,B 0,C 180,E1 -458.888,E2 -458.888} C_VEL
LIN {X 0,Y 608.485,Z 407.544,A -85,B 0,C 180,E1 -459.16,E2 -459.16} C_VEL
LIN {X 0,Y 608.477,Z 397.784,A -85,B 0,C 180,E1 -459.349,E2 -459.349} C_VEL
LIN {X 0,Y 608.473,Z 322.678,A -85,B 0,C 180,E1 -460.251,E2 -460.251} C_VEL
LIN {X 0,Y 608.452,Z 303.278,A -85,B 0,C 180,E1 -463.188,E2 -463.188} C_VEL
LIN {X 0,Y 608.491,Z 284.297,A -85,B 0,C 180,E1 -466.094,E2 -466.094} C_VEL
LIN {X 0,Y 608.512,Z 266.432,A -85,B 0,C 180,E1 -468.869,E2 -468.869} C_VEL
LIN {X 0,Y 608.483,Z 250.8,A -85,B 0,C 180,E1 -471.336,E2 -471.336} C_VEL
LIN {X 0,Y 608.415,Z 249.506,A -85,B 0,C 180,E1 -471.561,E2 -471.561} C_VEL
LIN {X 0,Y 608.406,Z 249.506,A -85,B 0,C 180,E1 -474.137,E2 -474.137} C_VEL
LIN {X 0,Y 608.435,Z 249.507,A -85,B 0,C 180,E1 -477.198,E2 -477.198} C_VEL
LIN {X 0,Y 608.396,Z 249.507,A -85,B 0,C 180,E1 -479.784,E2 -479.784} C_VEL
LIN {X 0,Y 608.421,Z 249.508,A -85,B 0,C 180,E1 -482.515,E2 -482.515} C_VEL
LIN {X 0,Y 608.409,Z 249.509,A -85,B 0,C 180,E1 -485.281,E2 -485.281} C_VEL
LIN {X 0,Y 608.399,Z 249.506,A -85,B 0,C 180,E1 -487.752,E2 -487.752} C_VEL
LIN {X 0,Y 608.412,Z 249.506,A -85,B 0,C 180,E1 -490.323,E2 -490.323} C_VEL
LIN {X 0,Y 608.479,Z 249.501,A -85,B 0,C 180,E1 -493.308,E2 -493.308} C_VEL
LIN {X 0,Y 608.427,Z 249.503,A -85,B 0,C 180,E1 -496.125,E2 -496.125} C_VEL
LIN {X 0,Y 608.443,Z 249.508,A -85,B 0,C 180,E1 -498.821,E2 -498.821} C_VEL
LIN {X 0,Y 608.445,Z 249.501,A -85,B 0,C 180,E1 -501.763,E2 -501.763} C_VEL
LIN {X 0,Y 608.441,Z 249.501,A -85,B 0,C 180,E1 -503.956,E2 -503.956} C_VEL
LIN {X 0,Y 608.422,Z 249.504,A -85,B 0,C 180,E1 -506.325,E2 -506.325} C_VEL
LIN {X 0,Y 608.448,Z 249.505,A -85,B 0,C 180,E1 -508.733,E2 -508.733} C_VEL
LIN {X 0,Y 608.481,Z 249.502,A -85,B 0,C 180,E1 -511.38,E2 -511.38} C_VEL
LIN {X 0,Y 608.452,Z 249.5,A -85,B 0,C 180,E1 -514.284,E2 -514.284} C_VEL
LIN {X 0,Y 608.443,Z 249.507,A -85,B 0,C 180,E1 -516.874,E2 -516.874} C_VEL
LIN {X 0,Y 608.463,Z 249.5,A -85,B 0,C 180,E1 -519.724,E2 -519.724} C_VEL
LIN {X 0,Y 608.447,Z 249.502,A -85,B 0,C 180,E1 -522.521,E2 -522.521} C_VEL
LIN {X 0,Y 608.47,Z 249.711,A -85,B 0,C 180,E1 -522.695,E2 -522.695} C_VEL
LIN {X 0,Y 608.455,Z 263.91,A -85,B 0,C 180,E1 -525.618,E2 -525.618} C_VEL
LIN {X 0,Y 608.439,Z 277.274,A -85,B 0,C 180,E1 -528.335,E2 -528.335} C_VEL
LIN {X 0,Y 608.428,Z 284.808,A -85,B 0,C 180,E1 -529.83,E2 -529.83} C_VEL
LIN {X 0,Y 608.465,Z 360.078,A -85,B 0,C 180,E1 -530.733,E2 -530.733} C_VEL
LIN {X 0,Y 608.426,Z 369.84,A -85,B 0,C 180,E1 -530.942,E2 -530.942} C_VEL
LIN {X 0,Y 608.437,Z 381.465,A -85,B 0,C 180,E1 -531.319,E2 -531.319} C_VEL
LIN {X 0,Y 608.464,Z 391.389,A -85,B 0,C 180,E1 -531.779,E2 -531.779} C_VEL
LIN {X 0,Y 608.475,Z 399.85,A -85,B 0,C 180,E1 -532.281,E2 -532.281} C_VEL
LIN {X 0,Y 608.462,Z 407.821,A -85,B 0,C 180,E1 -532.864,E2 -532.864} C_VEL
LIN {X 0,Y 608.47,Z 414.901,A -85,B 0,C 180,E1 -533.496,E2 -533.496} C_VEL
LIN {X 0,Y 608.459,Z 421.374,A -85,B 0,C 180,E1 -534.196,E2 -534.196} C_VEL
LIN {X 0,Y 608.436,Z 427.622,A -85,B 0,C 180,E1 -535.027,E2 -535.027} C_VEL
LIN {X 0,Y 608.432,Z 433.413,A -85,B 0,C 180,E1 -536.023,E2 -536.023} C_VEL
LIN {X 0,Y 608.447,Z 437.621,A -85,B 0,C 180,E1 -537.017,E2 -537.017} C_VEL
LIN {X 0,Y 608.439,Z 440.563,A -85,B 0,C 180,E1 -538.011,E2 -538.011} C_VEL
LIN {X 0,Y 608.448,Z 441.867,A -85,B 0,C 180,E1 -538.673,E2 -538.673} C_VEL
LIN {X 0,Y 608.434,Z 442.692,A -85,B 0,C 180,E1 -539.335,E2 -539.335} C_VEL
LIN {X 0,Y 608.432,Z 442.995,A -85,B 0,C 180,E1 -539.997,E2 -539.997} C_VEL
LIN {X 0,Y 608.437,Z 442.738,A -85,B 0,C 180,E1 -540.658,E2 -540.658} C_VEL
LIN {X 0,Y 608.447,Z 442.004,A -85,B 0,C 180,E1 -541.32,E2 -541.32} C_VEL
LIN {X 0,Y 608.443,Z 440.797,A -85,B 0,C 180,E1 -541.982,E2 -541.982} C_VEL
LIN {X 0,Y 608.446,Z 437.955,A -85,B 0,C 180,E1 -542.976,E2 -542.976} C_VEL
LIN {X 0,Y 608.444,Z 435.371,A -85,B 0,C 180,E1 -543.639,E2 -543.639} C_VEL
LIN {X 0,Y 608.447,Z 430.268,A -85,B 0,C 180,E1 -544.634,E2 -544.634} C_VEL
LIN {X 0,Y 608.461,Z 424.777,A -85,B 0,C 180,E1 -545.464,E2 -545.464} C_VEL
LIN {X 0,Y 608.454,Z 417.17,A -85,B 0,C 180,E1 -546.372,E2 -546.372} C_VEL
LIN {X 0,Y 608.461,Z 408.996,A -85,B 0,C 180,E1 -547.129,E2 -547.129} C_VEL
LIN {X 0,Y 608.458,Z 401.26,A -85,B 0,C 180,E1 -547.713,E2 -547.713} C_VEL
LIN {X 0,Y 608.471,Z 393.109,A -85,B 0,C 180,E1 -548.214,E2 -548.214} C_VEL
LIN {X 0,Y 608.48,Z 390,A -85,B 0,C 180,E1 -548.385,E2 -548.385} C_VEL
LIN {X 0,Y 607.796,Z 386.508,A -85,B 0,C 180,E1 -548.559,E2 -548.559} C_VEL
LIN {X 0,Y 604.928,Z 381.11,A -85,B 0,C 180,E1 -548.841,E2 -548.841} C_VEL
LIN {X 0,Y 602.109,Z 375.555,A -85,B 0,C 180,E1 -549.086,E2 -549.086} C_VEL
LIN {X 0,Y 601.485,Z 371.83,A -85,B 0,C 180,E1 -549.203,E2 -549.203} C_VEL
LIN {X 0,Y 601.498,Z 360.846,A -85,B 0,C 180,E1 -549.453,E2 -549.453} C_VEL
LIN {X 0,Y 601.524,Z 325.199,A -85,B 0,C 180,E1 -549.898,E2 -549.898} C_VEL
LIN {X 0,Y 601.36,Z 284.643,A -85,B 0,C 180,E1 -550.39,E2 -550.39} C_VEL
LIN {X 0,Y 601.404,Z 271.065,A -85,B 0,C 180,E1 -553.168,E2 -553.168} C_VEL
LIN {X 0,Y 601.382,Z 259.367,A -85,B 0,C 180,E1 -555.588,E2 -555.588} C_VEL
LIN {X 0,Y 601.362,Z 250.385,A -85,B 0,C 180,E1 -557.465,E2 -557.465} C_VEL
LIN {X 0,Y 601.358,Z 250.383,A -85,B 0,C 180,E1 -559.806,E2 -559.806} C_VEL
LIN {X 0,Y 601.387,Z 250.383,A -85,B 0,C 180,E1 -562.598,E2 -562.598} C_VEL
LIN {X 0,Y 601.378,Z 250.384,A -85,B 0,C 180,E1 -565.615,E2 -565.615} C_VEL
LIN {X 0,Y 601.34,Z 250.387,A -85,B 0,C 180,E1 -567.866,E2 -567.866} C_VEL
LIN {X 0,Y 601.35,Z 250.384,A -85,B 0,C 180,E1 -570.163,E2 -570.163} C_VEL
LIN {X 0,Y 601.37,Z 250.383,A -85,B 0,C 180,E1 -572.707,E2 -572.707} C_VEL
LIN {X 0,Y 601.357,Z 250.389,A -85,B 0,C 180,E1 -575.106,E2 -575.106} C_VEL
LIN {X 0,Y 601.402,Z 250.388,A -85,B 0,C 180,E1 -577.415,E2 -577.415} C_VEL
LIN {X 0,Y 601.359,Z 250.386,A -85,B 0,C 180,E1 -579.992,E2 -579.992} C_VEL
LIN {X 0,Y 601.335,Z 250.386,A -85,B 0,C 180,E1 -582.582,E2 -582.582} C_VEL
LIN {X 0,Y 601.36,Z 250.383,A -85,B 0,C 180,E1 -584.528,E2 -584.528} C_VEL
LIN {X 0,Y 601.381,Z 250.385,A -85,B 0,C 180,E1 -587.404,E2 -587.404} C_VEL
LIN {X 0,Y 601.373,Z 250.389,A -85,B 0,C 180,E1 -590.001,E2 -590.001} C_VEL
LIN {X 0,Y 601.386,Z 250.38,A -85,B 0,C 180,E1 -592.614,E2 -592.614} C_VEL
LIN {X 0,Y 601.346,Z 250.384,A -85,B 0,C 180,E1 -595.063,E2 -595.063} C_VEL
LIN {X 0,Y 601.378,Z 250.383,A -85,B 0,C 180,E1 -597.48,E2 -597.48} C_VEL
LIN {X 0,Y 601.402,Z 250.384,A -85,B 0,C 180,E1 -599.844,E2 -599.844} C_VEL
LIN {X 0,Y 601.39,Z 250.38,A -85,B 0,C 180,E1 -602.885,E2 -602.885} C_VEL
LIN {X 0,Y 601.349,Z 250.384,A -85,B 0,C 180,E1 -605.118,E2 -605.118} C_VEL
LIN {X 0,Y 601.359,Z 250.383,A -85,B 0,C 180,E1 -607.391,E2 -607.391} C_VEL
LIN {X 0,Y 601.365,Z 250.39,A -85,B 0,C 180,E1 -610.188,E2 -610.188} C_VEL
LIN {X 0,Y 601.38,Z 250.382,A -85,B 0,C 180,E1 -613.012,E2 -613.012} C_VEL
LIN {X 0,Y 601.358,Z 250.384,A -85,B 0,C 180,E1 -615.792,E2 -615.792} C_VEL
LIN {X 0,Y 601.392,Z 250.39,A -85,B 0,C 180,E1 -618.54,E2 -618.54} C_VEL
LIN {X 0,Y 601.385,Z 250.381,A -85,B 0,C 180,E1 -621.261,E2 -621.261} C_VEL
LIN {X 0,Y 601.391,Z 250.381,A -85,B 0,C 180,E1 -623.322,E2 -623.322} C_VEL
LIN {X 0,Y 601.373,Z 250.383,A -85,B 0,C 180,E1 -625.307,E2 -625.307} C_VEL
LIN {X 0,Y 601.394,Z 250.381,A -85,B 0,C 180,E1 -627.32,E2 -627.32} C_VEL
LIN {X 0,Y 601.373,Z 250.381,A -85,B 0,C 180,E1 -629.999,E2 -629.999} C_VEL
LIN {X 0,Y 601.402,Z 250.384,A -85,B 0,C 180,E1 -632.678,E2 -632.678} C_VEL
LIN {X 0,Y 601.404,Z 250.383,A -85,B 0,C 180,E1 -635.363,E2 -635.363} C_VEL
LIN {X 0,Y 601.377,Z 250.381,A -85,B 0,C 180,E1 -638.06,E2 -638.06} C_VEL
LIN {X 0,Y 601.375,Z 250.385,A -85,B 0,C 180,E1 -640.776,E2 -640.776} C_VEL
LIN {X 0,Y 601.39,Z 250.385,A -85,B 0,C 180,E1 -643.515,E2 -643.515} C_VEL
LIN {X 0,Y 601.372,Z 250.381,A -85,B 0,C 180,E1 -646.287,E2 -646.287} C_VEL
LIN {X 0,Y 601.367,Z 250.388,A -85,B 0,C 180,E1 -649.099,E2 -649.099} C_VEL
LIN {X 0,Y 601.378,Z 250.384,A -85,B 0,C 180,E1 -651.959,E2 -651.959} C_VEL
LIN {X 0,Y 601.384,Z 250.38,A -85,B 0,C 180,E1 -654.297,E2 -654.297} C_VEL
LIN {X 0,Y 601.359,Z 250.383,A -85,B 0,C 180,E1 -656.364,E2 -656.364} C_VEL
LIN {X 0,Y 601.374,Z 250.381,A -85,B 0,C 180,E1 -658.791,E2 -658.791} C_VEL
LIN {X 0,Y 601.388,Z 250.385,A -85,B 0,C 180,E1 -661.461,E2 -661.461} C_VEL
LIN {X 0,Y 601.386,Z 250.385,A -85,B 0,C 180,E1 -664.119,E2 -664.119} C_VEL
LIN {X 0,Y 601.353,Z 250.385,A -85,B 0,C 180,E1 -666.584,E2 -666.584} C_VEL
LIN {X 0,Y 601.38,Z 250.381,A -85,B 0,C 180,E1 -669.127,E2 -669.127} C_VEL
LIN {X 0,Y 601.395,Z 250.385,A -85,B 0,C 180,E1 -671.765,E2 -671.765} C_VEL
LIN {X 0,Y 601.375,Z 250.384,A -85,B 0,C 180,E1 -674.538,E2 -674.538} C_VEL
LIN {X 0,Y 601.356,Z 250.383,A -85,B 0,C 180,E1 -677.332,E2 -677.332} C_VEL
LIN {X 0,Y 601.367,Z 250.389,A -85,B 0,C 180,E1 -680.009,E2 -680.009} C_VEL
LIN {X 0,Y 601.391,Z 250.384,A -85,B 0,C 180,E1 -682.621,E2 -682.621} C_VEL
LIN {X 0,Y 601.383,Z 250.381,A -85,B 0,C 180,E1 -685.072,E2 -685.072} C_VEL
LIN {X 0,Y 601.368,Z 250.382,A -85,B 0,C 180,E1 -687.487,E2 -687.487} C_VEL
LIN {X 0,Y 601.361,Z 250.384,A -85,B 0,C 180,E1 -689.859,E2 -689.859} C_VEL
LIN {X 0,Y 601.393,Z 250.389,A -85,B 0,C 180,E1 -692.638,E2 -692.638} C_VEL
LIN {X 0,Y 601.369,Z 250.385,A -85,B 0,C 180,E1 -695.125,E2 -695.125} C_VEL
LIN {X 0,Y 601.38,Z 250.381,A -85,B 0,C 180,E1 -697.398,E2 -697.398} C_VEL
LIN {X 0,Y 601.366,Z 250.384,A -85,B 0,C 180,E1 -700.194,E2 -700.194} C_VEL
LIN {X 0,Y 601.402,Z 250.386,A -85,B 0,C 180,E1 -703.018,E2 -703.018} C_VEL
LIN {X 0,Y 601.347,Z 250.384,A -85,B 0,C 180,E1 -705.929,E2 -705.929} C_VEL
LIN {X 0,Y 601.403,Z 250.381,A -85,B 0,C 180,E1 -708.545,E2 -708.545} C_VEL
LIN {X 0,Y 601.414,Z 250.384,A -85,B 0,C 180,E1 -711.266,E2 -711.266} C_VEL
LIN {X 0,Y 601.359,Z 250.383,A -85,B 0,C 180,E1 -713.966,E2 -713.966} C_VEL
LIN {X 0,Y 601.354,Z 250.384,A -85,B 0,C 180,E1 -715.983,E2 -715.983} C_VEL
LIN {X 0,Y 601.377,Z 250.381,A -85,B 0,C 180,E1 -717.994,E2 -717.994} C_VEL
LIN {X 0,Y 601.4,Z 250.379,A -85,B 0,C 180,E1 -720.003,E2 -720.003} C_VEL
LIN {X 0,Y 601.389,Z 250.38,A -85,B 0,C 180,E1 -722.682,E2 -722.682} C_VEL
LIN {X 0,Y 601.409,Z 250.386,A -85,B 0,C 180,E1 -725.367,E2 -725.367} C_VEL
LIN {X 0,Y 601.417,Z 250.378,A -85,B 0,C 180,E1 -728.064,E2 -728.064} C_VEL
LIN {X 0,Y 601.384,Z 250.381,A -85,B 0,C 180,E1 -731.002,E2 -731.002} C_VEL
LIN {X 0,Y 601.392,Z 250.387,A -85,B 0,C 180,E1 -733.519,E2 -733.519} C_VEL
LIN {X 0,Y 601.399,Z 250.38,A -85,B 0,C 180,E1 -736.291,E2 -736.291} C_VEL
LIN {X 0,Y 601.39,Z 250.38,A -85,B 0,C 180,E1 -739.102,E2 -739.102} C_VEL
LIN {X 0,Y 601.382,Z 250.391,A -85,B 0,C 180,E1 -741.963,E2 -741.963} C_VEL
LIN {X 0,Y 601.431,Z 250.379,A -85,B 0,C 180,E1 -744.296,E2 -744.296} C_VEL
LIN {X 0,Y 601.366,Z 250.382,A -85,B 0,C 180,E1 -747.117,E2 -747.117} C_VEL
LIN {X 0,Y 601.372,Z 250.382,A -85,B 0,C 180,E1 -749.398,E2 -749.398} C_VEL
LIN {X 0,Y 601.387,Z 250.383,A -85,B 0,C 180,E1 -751.73,E2 -751.73} C_VEL
LIN {X 0,Y 601.4,Z 250.387,A -85,B 0,C 180,E1 -754.122,E2 -754.122} C_VEL
LIN {X 0,Y 601.378,Z 250.387,A -85,B 0,C 180,E1 -756.587,E2 -756.587} C_VEL
LIN {X 0,Y 601.372,Z 250.382,A -85,B 0,C 180,E1 -759.131,E2 -759.131} C_VEL
LIN {X 0,Y 601.393,Z 250.38,A -85,B 0,C 180,E1 -761.769,E2 -761.769} C_VEL
LIN {X 0,Y 601.392,Z 250.39,A -85,B 0,C 180,E1 -764.534,E2 -764.534} C_VEL
LIN {X 0,Y 601.424,Z 250.384,A -85,B 0,C 180,E1 -766.429,E2 -766.429} C_VEL
LIN {X 0,Y 601.38,Z 250.381,A -85,B 0,C 180,E1 -769.432,E2 -769.432} C_VEL
LIN {X 0,Y 601.374,Z 250.381,A -85,B 0,C 180,E1 -771.731,E2 -771.731} C_VEL
LIN {X 0,Y 601.353,Z 250.386,A -85,B 0,C 180,E1 -774.245,E2 -774.245} C_VEL
LIN {X 0,Y 601.397,Z 250.386,A -85,B 0,C 180,E1 -776.686,E2 -776.686} C_VEL
LIN {X 0,Y 601.396,Z 250.387,A -85,B 0,C 180,E1 -779.058,E2 -779.058} C_VEL
LIN {X 0,Y 601.416,Z 250.38,A -85,B 0,C 180,E1 -781.374,E2 -781.374} C_VEL
LIN {X 0,Y 601.379,Z 250.382,A -85,B 0,C 180,E1 -783.637,E2 -783.637} C_VEL
LIN {X 0,Y 601.415,Z 250.377,A -85,B 0,C 180,E1 -785.859,E2 -785.859} C_VEL
LIN {X 0,Y 601.385,Z 250.536,A -85,B 0,C 180,E1 -788.357,E2 -788.357} C_VEL
LIN {X 0,Y 601.534,Z 259.748,A -85,B 0,C 180,E1 -789.84,E2 -789.84} C_VEL
LIN {X 0,Y 601.493,Z 276.496,A -85,B 0,C 180,E1 -792.492,E2 -792.492} C_VEL
LIN {X 0,Y 601.442,Z 293.244,A -85,B 0,C 180,E1 -795.105,E2 -795.105} C_VEL
LIN {X 0,Y 601.429,Z 311.109,A -85,B 0,C 180,E1 -797.859,E2 -797.859} C_VEL
LIN {X 0,Y 601.4,Z 322.763,A -85,B 0,C 180,E1 -799.64,E2 -799.64} C_VEL
LIN {X 0,Y 601.503,Z 399.221,A -85,B 0,C 180,E1 -800.566,E2 -800.566} C_VEL
LIN {X 0,Y 601.477,Z 408.464,A -85,B 0,C 180,E1 -800.756,E2 -800.756} C_VEL
LIN {X 0,Y 601.439,Z 416.925,A -85,B 0,C 180,E1 -801.01,E2 -801.01} C_VEL
LIN {X 0,Y 601.443,Z 425.42,A -85,B 0,C 180,E1 -801.348,E2 -801.348} C_VEL
LIN {X 0,Y 601.449,Z 433.744,A -85,B 0,C 180,E1 -801.772,E2 -801.772} C_VEL
LIN {X 0,Y 601.424,Z 441.78,A -85,B 0,C 180,E1 -802.278,E2 -802.278} C_VEL
LIN {X 0,Y 601.413,Z 449.43,A -85,B 0,C 180,E1 -802.869,E2 -802.869} C_VEL
LIN {X 0,Y 601.394,Z 457.164,A -85,B 0,C 180,E1 -803.598,E2 -803.598} C_VEL
LIN {X 0,Y 601.383,Z 464.439,A -85,B 0,C 180,E1 -804.469,E2 -804.469} C_VEL
LIN {X 0,Y 601.341,Z 469.992,A -85,B 0,C 180,E1 -805.309,E2 -805.309} C_VEL
LIN {X 0,Y 601.365,Z 475.152,A -85,B 0,C 180,E1 -806.316,E2 -806.316} C_VEL
LIN {X 0,Y 601.343,Z 477.791,A -85,B 0,C 180,E1 -806.986,E2 -806.986} C_VEL
LIN {X 0,Y 601.343,Z 480.682,A -85,B 0,C 180,E1 -807.992,E2 -807.992} C_VEL
LIN {X 0,Y 601.345,Z 481.936,A -85,B 0,C 180,E1 -808.662,E2 -808.662} C_VEL
LIN {X 0,Y 601.335,Z 482.714,A -85,B 0,C 180,E1 -809.331,E2 -809.331} C_VEL
LIN {X 0,Y 601.332,Z 483,A -85,B 0,C 180,E1 -810.001,E2 -810.001} C_VEL
LIN {X 0,Y 601.335,Z 482.713,A -85,B 0,C 180,E1 -810.671,E2 -810.671} C_VEL
LIN {X 0,Y 601.345,Z 481.933,A -85,B 0,C 180,E1 -811.34,E2 -811.34} C_VEL
LIN {X 0,Y 601.343,Z 480.676,A -85,B 0,C 180,E1 -812.01,E2 -812.01} C_VEL
LIN {X 0,Y 601.343,Z 477.783,A -85,B 0,C 180,E1 -813.016,E2 -813.016} C_VEL
LIN {X 0,Y 601.365,Z 475.142,A -85,B 0,C 180,E1 -813.686,E2 -813.686} C_VEL
LIN {X 0,Y 601.341,Z 469.979,A -85,B 0,C 180,E1 -814.694,E2 -814.694} C_VEL
LIN {X 0,Y 601.383,Z 464.422,A -85,B 0,C 180,E1 -815.534,E2 -815.534} C_VEL
LIN {X 0,Y 601.394,Z 457.161,A -85,B 0,C 180,E1 -816.402,E2 -816.402} C_VEL
LIN {X 0,Y 601.414,Z 449.404,A -85,B 0,C 180,E1 -817.133,E2 -817.133} C_VEL
LIN {X 0,Y 601.401,Z 441.748,A -85,B 0,C 180,E1 -817.724,E2 -817.724} C_VEL
LIN {X 0,Y 601.45,Z 433.704,A -85,B 0,C 180,E1 -818.231,E2 -818.231} C_VEL
LIN {X 0,Y 601.443,Z 425.37,A -85,B 0,C 180,E1 -818.654,E2 -818.654} C_VEL
LIN {X 0,Y 601.44,Z 416.861,A -85,B 0,C 180,E1 -818.993,E2 -818.993} C_VEL
LIN {X 0,Y 601.465,Z 406.714,A -85,B 0,C 180,E1 -819.289,E2 -819.289} C_VEL
LIN {X 0,Y 601.499,Z 394.973,A -85,B 0,C 180,E1 -819.5,E2 -819.5} C_VEL
LIN {X 0,Y 601.405,Z 322.678,A -85,B 0,C 180,E1 -820.373,E2 -820.373} C_VEL
LIN {X 0,Y 601.434,Z 304.395,A -85,B 0,C 180,E1 -823.172,E2 -823.172} C_VEL
LIN {X 0,Y 601.472,Z 285.413,A -85,B 0,C 180,E1 -826.113,E2 -826.113} C_VEL
LIN {X 0,Y 601.53,Z 267.988,A -85,B 0,C 180,E1 -828.85,E2 -828.85} C_VEL
LIN {X 0,Y 601.517,Z 251.917,A -85,B 0,C 180,E1 -831.416,E2 -831.416} C_VEL
LIN {X 0,Y 601.383,Z 250.384,A -85,B 0,C 180,E1 -831.691,E2 -831.691} C_VEL
LIN {X 0,Y 601.38,Z 250.383,A -85,B 0,C 180,E1 -834.28,E2 -834.28} C_VEL
LIN {X 0,Y 601.378,Z 250.384,A -85,B 0,C 180,E1 -837.354,E2 -837.354} C_VEL
LIN {X 0,Y 601.36,Z 250.386,A -85,B 0,C 180,E1 -839.397,E2 -839.397} C_VEL
LIN {X 0,Y 601.364,Z 250.383,A -85,B 0,C 180,E1 -841.73,E2 -841.73} C_VEL
LIN {X 0,Y 601.34,Z 250.386,A -85,B 0,C 180,E1 -844.125,E2 -844.125} C_VEL
LIN {X 0,Y 601.385,Z 250.385,A -85,B 0,C 180,E1 -846.585,E2 -846.585} C_VEL
LIN {X 0,Y 601.396,Z 250.38,A -85,B 0,C 180,E1 -849.529,E2 -849.529} C_VEL
LIN {X 0,Y 601.381,Z 250.381,A -85,B 0,C 180,E1 -851.77,E2 -851.77} C_VEL
LIN {X 0,Y 601.38,Z 250.384,A -85,B 0,C 180,E1 -854.529,E2 -854.529} C_VEL
LIN {X 0,Y 601.384,Z 250.385,A -85,B 0,C 180,E1 -857.326,E2 -857.326} C_VEL
LIN {X 0,Y 601.383,Z 250.38,A -85,B 0,C 180,E1 -860.001,E2 -860.001} C_VEL
LIN {X 0,Y 601.407,Z 250.381,A -85,B 0,C 180,E1 -862.622,E2 -862.622} C_VEL
LIN {X 0,Y 601.413,Z 250.387,A -85,B 0,C 180,E1 -865.066,E2 -865.066} C_VEL
LIN {X 0,Y 601.44,Z 250.377,A -85,B 0,C 180,E1 -867.483,E2 -867.483} C_VEL
LIN {X 0,Y 601.414,Z 250.377,A -85,B 0,C 180,E1 -869.855,E2 -869.855} C_VEL
LIN {X 0,Y 601.385,Z 250.38,A -85,B 0,C 180,E1 -872.129,E2 -872.129} C_VEL
LIN {X 0,Y 601.4,Z 250.379,A -85,B 0,C 180,E1 -874.379,E2 -874.379} C_VEL
LIN {X 0,Y 601.393,Z 250.382,A -85,B 0,C 180,E1 -876.586,E2 -876.586} C_VEL
LIN {X 0,Y 601.435,Z 250.379,A -85,B 0,C 180,E1 -879.476,E2 -879.476} C_VEL
LIN {X 0,Y 601.395,Z 250.379,A -85,B 0,C 180,E1 -882.309,E2 -882.309} C_VEL
LIN {X 0,Y 601.422,Z 250.549,A -85,B 0,C 180,E1 -882.661,E2 -882.661} C_VEL
LIN {X 0,Y 601.394,Z 263.912,A -85,B 0,C 180,E1 -885.446,E2 -885.446} C_VEL
LIN {X 0,Y 601.387,Z 275.606,A -85,B 0,C 180,E1 -887.854,E2 -887.854} C_VEL
LIN {X 0,Y 601.36,Z 284.854,A -85,B 0,C 180,E1 -889.71,E2 -889.71} C_VEL
LIN {X 0,Y 601.46,Z 360.112,A -85,B 0,C 180,E1 -890.624,E2 -890.624} C_VEL
LIN {X 0,Y 601.431,Z 369.865,A -85,B 0,C 180,E1 -890.836,E2 -890.836} C_VEL
LIN {X 0,Y 601.405,Z 381.478,A -85,B 0,C 180,E1 -891.217,E2 -891.217} C_VEL
LIN {X 0,Y 601.446,Z 391.412,A -85,B 0,C 180,E1 -891.683,E2 -891.683} C_VEL
LIN {X 0,Y 601.434,Z 399.872,A -85,B 0,C 180,E1 -892.19,E2 -892.19} C_VEL
LIN {X 0,Y 601.415,Z 407.835,A -85,B 0,C 180,E1 -892.78,E2 -892.78} C_VEL
LIN {X 0,Y 601.416,Z 415.154,A -85,B 0,C 180,E1 -893.443,E2 -893.443} C_VEL
LIN {X 0,Y 601.392,Z 422.802,A -85,B 0,C 180,E1 -894.296,E2 -894.296} C_VEL
LIN {X 0,Y 601.365,Z 429.72,A -85,B 0,C 180,E1 -895.304,E2 -895.304} C_VEL
LIN {X 0,Y 601.365,Z 434.941,A -85,B 0,C 180,E1 -896.311,E2 -896.311} C_VEL
LIN {X 0,Y 601.326,Z 438.774,A -85,B 0,C 180,E1 -897.317,E2 -897.317} C_VEL
LIN {X 0,Y 601.338,Z 440.571,A -85,B 0,C 180,E1 -897.987,E2 -897.987} C_VEL
LIN {X 0,Y 601.348,Z 441.875,A -85,B 0,C 180,E1 -898.657,E2 -898.657} C_VEL
LIN {X 0,Y 601.335,Z 442.698,A -85,B 0,C 180,E1 -899.327,E2 -899.327} C_VEL
LIN {X 0,Y 601.333,Z 442.995,A -85,B 0,C 180,E1 -899.997,E2 -899.997} C_VEL
LIN {X 0,Y 601.338,Z 442.743,A -85,B 0,C 180,E1 -900.666,E2 -900.666} C_VEL
LIN {X 0,Y 601.346,Z 442.011,A -85,B 0,C 180,E1 -901.336,E2 -901.336} C_VEL
LIN {X 0,Y 601.342,Z 440.802,A -85,B 0,C 180,E1 -902.006,E2 -902.006} C_VEL
LIN {X 0,Y 601.345,Z 437.959,A -85,B 0,C 180,E1 -903.011,E2 -903.011} C_VEL
LIN {X 0,Y 601.344,Z 433.862,A -85,B 0,C 180,E1 -904.017,E2 -904.017} C_VEL
LIN {X 0,Y 601.346,Z 428.29,A -85,B 0,C 180,E1 -905.025,E2 -905.025} C_VEL
LIN {X 0,Y 601.385,Z 422.207,A -85,B 0,C 180,E1 -905.865,E2 -905.865} C_VEL
LIN {X 0,Y 601.414,Z 415.254,A -85,B 0,C 180,E1 -906.637,E2 -906.637} C_VEL
LIN {X 0,Y 601.405,Z 407.983,A -85,B 0,C 180,E1 -907.297,E2 -907.297} C_VEL
LIN {X 0,Y 601.441,Z 398.827,A -85,B 0,C 180,E1 -907.972,E2 -907.972} C_VEL
LIN {X 0,Y 601.446,Z 388.324,A -85,B 0,C 180,E1 -908.564,E2 -908.564} C_VEL
LIN {X 0,Y 601.458,Z 378.284,A -85,B 0,C 180,E1 -908.987,E2 -908.987} C_VEL
LIN {X 0,Y 601.485,Z 371.83,A -85,B 0,C 180,E1 -909.203,E2 -909.203} C_VEL
LIN {X 0,Y 601.058,Z 366.149,A -85,B 0,C 180,E1 -909.358,E2 -909.358} C_VEL
LIN {X 0,Y 599.536,Z 360.577,A -85,B 0,C 180,E1 -909.492,E2 -909.492} C_VEL
LIN {X 0,Y 595.248,Z 347.592,A -85,B 0,C 180,E1 -909.738,E2 -909.738} C_VEL
LIN {X 0,Y 594.513,Z 341.784,A -85,B 0,C 180,E1 -909.817,E2 -909.817} C_VEL
LIN {X 0,Y 594.426,Z 285.798,A -85,B 0,C 180,E1 -910.491,E2 -910.491} C_VEL
LIN {X 0,Y 594.288,Z 284.64,A -85,B 0,C 180,E1 -910.515,E2 -910.515} C_VEL
LIN {X 0,Y 594.36,Z 271.063,A -85,B 0,C 180,E1 -913.327,E2 -913.327} C_VEL
LIN {X 0,Y 594.338,Z 257.693,A -85,B 0,C 180,E1 -916.13,E2 -916.13} C_VEL
LIN {X 0,Y 594.326,Z 251.262,A -85,B 0,C 180,E1 -917.501,E2 -917.501} C_VEL
LIN {X 0,Y 594.33,Z 251.259,A -85,B 0,C 180,E1 -920.05,E2 -920.05} C_VEL
LIN {X 0,Y 594.33,Z 251.268,A -85,B 0,C 180,E1 -922.964,E2 -922.964} C_VEL
LIN {X 0,Y 594.32,Z 251.26,A -85,B 0,C 180,E1 -925.941,E2 -925.941} C_VEL
LIN {X 0,Y 594.298,Z 251.263,A -85,B 0,C 180,E1 -928.225,E2 -928.225} C_VEL
LIN {X 0,Y 594.33,Z 251.259,A -85,B 0,C 180,E1 -930.557,E2 -930.557} C_VEL
LIN {X 0,Y 594.348,Z 251.261,A -85,B 0,C 180,E1 -932.946,E2 -932.946} C_VEL
LIN {X 0,Y 594.318,Z 251.271,A -85,B 0,C 180,E1 -935.405,E2 -935.405} C_VEL
LIN {X 0,Y 594.341,Z 251.261,A -85,B 0,C 180,E1 -937.937,E2 -937.937} C_VEL
LIN {X 0,Y 594.334,Z 251.259,A -85,B 0,C 180,E1 -940.816,E2 -940.816} C_VEL
LIN {X 0,Y 594.324,Z 251.267,A -85,B 0,C 180,E1 -943.834,E2 -943.834} C_VEL
LIN {X 0,Y 594.326,Z 251.259,A -85,B 0,C 180,E1 -946.696,E2 -946.696} C_VEL
LIN {X 0,Y 594.342,Z 251.262,A -85,B 0,C 180,E1 -949.43,E2 -949.43} C_VEL
LIN {X 0,Y 594.348,Z 251.259,A -85,B 0,C 180,E1 -952.387,E2 -952.387} C_VEL
LIN {X 0,Y 594.305,Z 251.262,A -85,B 0,C 180,E1 -954.672,E2 -954.672} C_VEL
LIN {X 0,Y 594.329,Z 251.259,A -85,B 0,C 180,E1 -957.085,E2 -957.085} C_VEL
LIN {X 0,Y 594.35,Z 251.26,A -85,B 0,C 180,E1 -959.666,E2 -959.666} C_VEL
LIN {X 0,Y 594.321,Z 251.264,A -85,B 0,C 180,E1 -962.536,E2 -962.536} C_VEL
LIN {X 0,Y 594.342,Z 251.259,A -85,B 0,C 180,E1 -964.805,E2 -964.805} C_VEL
LIN {X 0,Y 594.311,Z 251.261,A -85,B 0,C 180,E1 -967.261,E2 -967.261} C_VEL
LIN {X 0,Y 594.325,Z 251.263,A -85,B 0,C 180,E1 -969.944,E2 -969.944} C_VEL
LIN {X 0,Y 594.34,Z 251.262,A -85,B 0,C 180,E1 -972.804,E2 -972.804} C_VEL
LIN {X 0,Y 594.328,Z 251.26,A -85,B 0,C 180,E1 -975.823,E2 -975.823} C_VEL
LIN {X 0,Y 594.386,Z 251.257,A -85,B 0,C 180,E1 -978.894,E2 -978.894} C_VEL
LIN {X 0,Y 594.356,Z 251.256,A -85,B 0,C 180,E1 -981.841,E2 -981.841} C_VEL
LIN {X 0,Y 594.37,Z 251.262,A -85,B 0,C 180,E1 -984.571,E2 -984.571} C_VEL
LIN {X 0,Y 594.36,Z 251.258,A -85,B 0,C 180,E1 -987.288,E2 -987.288} C_VEL
LIN {X 0,Y 594.342,Z 251.257,A -85,B 0,C 180,E1 -989.999,E2 -989.999} C_VEL
LIN {X 0,Y 594.367,Z 251.261,A -85,B 0,C 180,E1 -992.71,E2 -992.71} C_VEL
LIN {X 0,Y 594.361,Z 251.259,A -85,B 0,C 180,E1 -995.427,E2 -995.427} C_VEL
LIN {X 0,Y 594.355,Z 251.256,A -85,B 0,C 180,E1 -998.156,E2 -998.156} C_VEL
LIN {X 0,Y 594.388,Z 251.261,A -85,B 0,C 180,E1 -1001.107,E2 -1001.107} C_VEL
LIN {X 0,Y 594.324,Z 251.259,A -85,B 0,C 180,E1 -1004.175,E2 -1004.175} C_VEL
LIN {X 0,Y 594.347,Z 251.265,A -85,B 0,C 180,E1 -1007.193,E2 -1007.193} C_VEL
LIN {X 0,Y 594.324,Z 251.261,A -85,B 0,C 180,E1 -1010.054,E2 -1010.054} C_VEL
LIN {X 0,Y 594.304,Z 251.262,A -85,B 0,C 180,E1 -1012.738,E2 -1012.738} C_VEL
LIN {X 0,Y 594.342,Z 251.262,A -85,B 0,C 180,E1 -1015.193,E2 -1015.193} C_VEL
LIN {X 0,Y 594.324,Z 251.269,A -85,B 0,C 180,E1 -1017.529,E2 -1017.529} C_VEL
LIN {X 0,Y 594.342,Z 251.259,A -85,B 0,C 180,E1 -1020.333,E2 -1020.333} C_VEL
LIN {X 0,Y 594.322,Z 251.26,A -85,B 0,C 180,E1 -1022.952,E2 -1022.952} C_VEL
LIN {X 0,Y 594.328,Z 251.263,A -85,B 0,C 180,E1 -1025.408,E2 -1025.408} C_VEL
LIN {X 0,Y 594.348,Z 251.267,A -85,B 0,C 180,E1 -1027.941,E2 -1027.941} C_VEL
LIN {X 0,Y 594.339,Z 251.258,A -85,B 0,C 180,E1 -1030.827,E2 -1030.827} C_VEL
LIN {X 0,Y 594.333,Z 251.259,A -85,B 0,C 180,E1 -1033.3,E2 -1033.3} C_VEL
LIN {X 0,Y 594.332,Z 251.269,A -85,B 0,C 180,E1 -1036.162,E2 -1036.162} C_VEL
LIN {X 0,Y 594.329,Z 251.259,A -85,B 0,C 180,E1 -1039.181,E2 -1039.181} C_VEL
LIN {X 0,Y 594.34,Z 251.257,A -85,B 0,C 180,E1 -1041.298,E2 -1041.298} C_VEL
LIN {X 0,Y 594.349,Z 251.258,A -85,B 0,C 180,E1 -1043.762,E2 -1043.762} C_VEL
LIN {X 0,Y 594.356,Z 251.264,A -85,B 0,C 180,E1 -1046.244,E2 -1046.244} C_VEL
LIN {X 0,Y 594.35,Z 251.264,A -85,B 0,C 180,E1 -1048.655,E2 -1048.655} C_VEL
LIN {X 0,Y 594.34,Z 251.26,A -85,B 0,C 180,E1 -1051.046,E2 -1051.046} C_VEL
LIN {X 0,Y 594.35,Z 251.257,A -85,B 0,C 180,E1 -1053.304,E2 -1053.304} C_VEL
LIN {X 0,Y 594.314,Z 251.261,A -85,B 0,C 180,E1 -1055.578,E2 -1055.578} C_VEL
LIN {X 0,Y 594.317,Z 251.26,A -85,B 0,C 180,E1 -1057.77,E2 -1057.77} C_VEL
LIN {X 0,Y 594.332,Z 251.259,A -85,B 0,C 180,E1 -1059.95,E2 -1059.95} C_VEL
LIN {X 0,Y 594.358,Z 251.266,A -85,B 0,C 180,E1 -1062.81,E2 -1062.81} C_VEL
LIN {X 0,Y 594.333,Z 251.258,A -85,B 0,C 180,E1 -1065.84,E2 -1065.84} C_VEL
LIN {X 0,Y 594.373,Z 251.263,A -85,B 0,C 180,E1 -1068.925,E2 -1068.925} C_VEL
LIN {X 0,Y 594.331,Z 251.259,A -85,B 0,C 180,E1 -1071.846,E2 -1071.846} C_VEL
LIN {X 0,Y 594.319,Z 251.261,A -85,B 0,C 180,E1 -1073.894,E2 -1073.894} C_VEL
LIN {X 0,Y 594.311,Z 251.262,A -85,B 0,C 180,E1 -1075.935,E2 -1075.935} C_VEL
LIN {X 0,Y 594.351,Z 251.257,A -85,B 0,C 180,E1 -1077.971,E2 -1077.971} C_VEL
LIN {X 0,Y 594.371,Z 251.255,A -85,B 0,C 180,E1 -1080.003,E2 -1080.003} C_VEL
LIN {X 0,Y 594.36,Z 251.256,A -85,B 0,C 180,E1 -1082.714,E2 -1082.714} C_VEL
LIN {X 0,Y 594.372,Z 251.264,A -85,B 0,C 180,E1 -1085.431,E2 -1085.431} C_VEL
LIN {X 0,Y 594.359,Z 251.257,A -85,B 0,C 180,E1 -1088.16,E2 -1088.16} C_VEL
LIN {X 0,Y 594.351,Z 251.258,A -85,B 0,C 180,E1 -1091.064,E2 -1091.064} C_VEL
LIN {X 0,Y 594.36,Z 251.266,A -85,B 0,C 180,E1 -1093.682,E2 -1093.682} C_VEL
LIN {X 0,Y 594.32,Z 251.26,A -85,B 0,C 180,E1 -1096.702,E2 -1096.702} C_VEL
LIN {X 0,Y 594.344,Z 251.26,A -85,B 0,C 180,E1 -1099.338,E2 -1099.338} C_VEL
LIN {X 0,Y 594.337,Z 251.262,A -85,B 0,C 180,E1 -1101.507,E2 -1101.507} C_VEL
LIN {X 0,Y 594.38,Z 251.256,A -85,B 0,C 180,E1 -1104.449,E2 -1104.449} C_VEL
LIN {X 0,Y 594.334,Z 251.259,A -85,B 0,C 180,E1 -1106.704,E2 -1106.704} C_VEL
LIN {X 0,Y 594.362,Z 251.255,A -85,B 0,C 180,E1 -1109.002,E2 -1109.002} C_VEL
LIN {X 0,Y 594.361,Z 251.257,A -85,B 0,C 180,E1 -1111.644,E2 -1111.644} C_VEL
LIN {X 0,Y 594.353,Z 251.265,A -85,B 0,C 180,E1 -1114.138,E2 -1114.138} C_VEL
LIN {X 0,Y 594.319,Z 251.261,A -85,B 0,C 180,E1 -1117.093,E2 -1117.093} C_VEL
LIN {X 0,Y 594.332,Z 251.26,A -85,B 0,C 180,E1 -1119.772,E2 -1119.772} C_VEL
LIN {X 0,Y 594.355,Z 251.265,A -85,B 0,C 180,E1 -1122.378,E2 -1122.378} C_VEL
LIN {X 0,Y 594.309,Z 251.263,A -85,B 0,C 180,E1 -1125.198,E2 -1125.198} C_VEL
LIN {X 0,Y 594.324,Z 251.259,A -85,B 0,C 180,E1 -1127.623,E2 -1127.623} C_VEL
LIN {X 0,Y 594.352,Z 251.261,A -85,B 0,C 180,E1 -1130.32,E2 -1130.32} C_VEL
LIN {X 0,Y 594.376,Z 251.261,A -85,B 0,C 180,E1 -1132.915,E2 -1132.915} C_VEL
LIN {X 0,Y 594.351,Z 251.256,A -85,B 0,C 180,E1 -1135.867,E2 -1135.867} C_VEL
LIN {X 0,Y 594.341,Z 251.264,A -85,B 0,C 180,E1 -1138.65,E2 -1138.65} C_VEL
LIN {X 0,Y 594.375,Z 251.263,A -85,B 0,C 180,E1 -1141.045,E2 -1141.045} C_VEL
LIN {X 0,Y 594.335,Z 251.258,A -85,B 0,C 180,E1 -1144.056,E2 -1144.056} C_VEL
LIN {X 0,Y 594.345,Z 251.258,A -85,B 0,C 180,E1 -1146.296,E2 -1146.296} C_VEL
LIN {X 0,Y 594.357,Z 251.374,A -85,B 0,C 180,E1 -1148.225,E2 -1148.225} C_VEL
LIN {X 0,Y 594.567,Z 259.748,A -85,B 0,C 180,E1 -1149.594,E2 -1149.594} C_VEL
LIN {X 0,Y 594.516,Z 275.379,A -85,B 0,C 180,E1 -1152.102,E2 -1152.102} C_VEL
LIN {X 0,Y 594.395,Z 292.128,A -85,B 0,C 180,E1 -1154.749,E2 -1154.749} C_VEL
LIN {X 0,Y 594.392,Z 311.109,A -85,B 0,C 180,E1 -1157.713,E2 -1157.713} C_VEL
LIN {X 0,Y 594.352,Z 322.763,A -85,B 0,C 180,E1 -1159.516,E2 -1159.516} C_VEL
LIN {X 0,Y 594.548,Z 357.604,A -85,B 0,C 180,E1 -1159.939,E2 -1159.939} C_VEL
LIN {X 0,Y 594.498,Z 400.519,A -85,B 0,C 180,E1 -1160.475,E2 -1160.475} C_VEL
LIN {X 0,Y 594.45,Z 410.955,A -85,B 0,C 180,E1 -1160.71,E2 -1160.71} C_VEL
LIN {X 0,Y 594.425,Z 423.561,A -85,B 0,C 180,E1 -1161.16,E2 -1161.16} C_VEL
LIN {X 0,Y 594.417,Z 432.259,A -85,B 0,C 180,E1 -1161.588,E2 -1161.588} C_VEL
LIN {X 0,Y 594.374,Z 440.564,A -85,B 0,C 180,E1 -1162.101,E2 -1162.101} C_VEL
LIN {X 0,Y 594.351,Z 448.417,A -85,B 0,C 180,E1 -1162.698,E2 -1162.698} C_VEL
LIN {X 0,Y 594.343,Z 455.528,A -85,B 0,C 180,E1 -1163.358,E2 -1163.358} C_VEL
LIN {X 0,Y 594.318,Z 463.2,A -85,B 0,C 180,E1 -1164.232,E2 -1164.232} C_VEL
LIN {X 0,Y 594.289,Z 469.035,A -85,B 0,C 180,E1 -1165.083,E2 -1165.083} C_VEL
LIN {X 0,Y 594.261,Z 473.636,A -85,B 0,C 180,E1 -1165.932,E2 -1165.932} C_VEL
LIN {X 0,Y 594.267,Z 476.626,A -85,B 0,C 180,E1 -1166.611,E2 -1166.611} C_VEL
LIN {X 0,Y 594.228,Z 478.937,A -85,B 0,C 180,E1 -1167.29,E2 -1167.29} C_VEL
LIN {X 0,Y 594.242,Z 480.682,A -85,B 0,C 180,E1 -1167.968,E2 -1167.968} C_VEL
LIN {X 0,Y 594.245,Z 481.937,A -85,B 0,C 180,E1 -1168.646,E2 -1168.646} C_VEL
LIN {X 0,Y 594.235,Z 482.713,A -85,B 0,C 180,E1 -1169.324,E2 -1169.324} C_VEL
LIN {X 0,Y 594.233,Z 483,A -85,B 0,C 180,E1 -1170.001,E2 -1170.001} C_VEL
LIN {X 0,Y 594.235,Z 482.712,A -85,B 0,C 180,E1 -1170.679,E2 -1170.679} C_VEL
LIN {X 0,Y 594.245,Z 481.934,A -85,B 0,C 180,E1 -1171.357,E2 -1171.357} C_VEL
LIN {X 0,Y 594.242,Z 480.677,A -85,B 0,C 180,E1 -1172.034,E2 -1172.034} C_VEL
LIN {X 0,Y 594.246,Z 477.783,A -85,B 0,C 180,E1 -1173.052,E2 -1173.052} C_VEL
LIN {X 0,Y 594.286,Z 475.142,A -85,B 0,C 180,E1 -1173.73,E2 -1173.73} C_VEL
LIN {X 0,Y 594.256,Z 469.979,A -85,B 0,C 180,E1 -1174.75,E2 -1174.75} C_VEL
LIN {X 0,Y 594.318,Z 463.18,A -85,B 0,C 180,E1 -1175.77,E2 -1175.77} C_VEL
LIN {X 0,Y 594.344,Z 455.513,A -85,B 0,C 180,E1 -1176.644,E2 -1176.644} C_VEL
LIN {X 0,Y 594.352,Z 448.391,A -85,B 0,C 180,E1 -1177.304,E2 -1177.304} C_VEL
LIN {X 0,Y 594.375,Z 440.533,A -85,B 0,C 180,E1 -1177.902,E2 -1177.902} C_VEL
LIN {X 0,Y 594.431,Z 430.719,A -85,B 0,C 180,E1 -1178.5,E2 -1178.5} C_VEL
LIN {X 0,Y 594.439,Z 419.269,A -85,B 0,C 180,E1 -1179.014,E2 -1179.014} C_VEL
LIN {X 0,Y 594.458,Z 409.205,A -85,B 0,C 180,E1 -1179.335,E2 -1179.335} C_VEL
LIN {X 0,Y 594.499,Z 400.382,A -85,B 0,C 180,E1 -1179.528,E2 -1179.528} C_VEL
LIN {X 0,Y 594.399,Z 323.426,A -85,B 0,C 180,E1 -1180.475,E2 -1180.475} C_VEL
LIN {X 0,Y 594.341,Z 322.539,A -85,B 0,C 180,E1 -1180.519,E2 -1180.519} C_VEL
LIN {X 0,Y 594.378,Z 304.395,A -85,B 0,C 180,E1 -1183.332,E2 -1183.332} C_VEL
LIN {X 0,Y 594.489,Z 285.413,A -85,B 0,C 180,E1 -1186.307,E2 -1186.307} C_VEL
LIN {X 0,Y 594.587,Z 266.432,A -85,B 0,C 180,E1 -1189.328,E2 -1189.328} C_VEL
LIN {X 0,Y 594.552,Z 253.033,A -85,B 0,C 180,E1 -1191.497,E2 -1191.497} C_VEL
LIN {X 0,Y 594.344,Z 251.262,A -85,B 0,C 180,E1 -1191.824,E2 -1191.824} C_VEL
LIN {X 0,Y 594.345,Z 251.262,A -85,B 0,C 180,E1 -1194.449,E2 -1194.449} C_VEL
LIN {X 0,Y 594.332,Z 251.261,A -85,B 0,C 180,E1 -1197.515,E2 -1197.515} C_VEL
LIN {X 0,Y 594.312,Z 251.262,A -85,B 0,C 180,E1 -1199.781,E2 -1199.781} C_VEL
LIN {X 0,Y 594.334,Z 251.259,A -85,B 0,C 180,E1 -1202.15,E2 -1202.15} C_VEL
LIN {X 0,Y 594.314,Z 251.265,A -85,B 0,C 180,E1 -1205.317,E2 -1205.317} C_VEL
LIN {X 0,Y 594.306,Z 251.262,A -85,B 0,C 180,E1 -1207.948,E2 -1207.948} C_VEL
LIN {X 0,Y 594.365,Z 251.263,A -85,B 0,C 180,E1 -1210.819,E2 -1210.819} C_VEL
LIN {X 0,Y 594.344,Z 251.257,A -85,B 0,C 180,E1 -1213.835,E2 -1213.835} C_VEL
LIN {X 0,Y 594.35,Z 251.262,A -85,B 0,C 180,E1 -1216.697,E2 -1216.697} C_VEL
LIN {X 0,Y 594.366,Z 251.258,A -85,B 0,C 180,E1 -1219.431,E2 -1219.431} C_VEL
LIN {X 0,Y 594.367,Z 251.255,A -85,B 0,C 180,E1 -1222.395,E2 -1222.395} C_VEL
LIN {X 0,Y 594.381,Z 251.257,A -85,B 0,C 180,E1 -1225.418,E2 -1225.418} C_VEL
LIN {X 0,Y 594.38,Z 251.254,A -85,B 0,C 180,E1 -1228.358,E2 -1228.358} C_VEL
LIN {X 0,Y 594.389,Z 251.262,A -85,B 0,C 180,E1 -1231.042,E2 -1231.042} C_VEL
LIN {X 0,Y 594.35,Z 251.257,A -85,B 0,C 180,E1 -1234.053,E2 -1234.053} C_VEL
LIN {X 0,Y 594.377,Z 251.254,A -85,B 0,C 180,E1 -1236.293,E2 -1236.293} C_VEL
LIN {X 0,Y 594.41,Z 251.259,A -85,B 0,C 180,E1 -1239.222,E2 -1239.222} C_VEL
LIN {X 0,Y 594.35,Z 251.257,A -85,B 0,C 180,E1 -1242.092,E2 -1242.092} C_VEL
LIN {X 0,Y 594.394,Z 251.387,A -85,B 0,C 180,E1 -1242.627,E2 -1242.627} C_VEL
LIN {X 0,Y 594.342,Z 263.915,A -85,B 0,C 180,E1 -1245.269,E2 -1245.269} C_VEL
LIN {X 0,Y 594.321,Z 275.609,A -85,B 0,C 180,E1 -1247.708,E2 -1247.708} C_VEL
LIN {X 0,Y 594.272,Z 284.9,A -85,B 0,C 180,E1 -1249.585,E2 -1249.585} C_VEL
LIN {X 0,Y 594.567,Z 292.051,A -85,B 0,C 180,E1 -1249.677,E2 -1249.677} C_VEL
LIN {X 0,Y 594.47,Z 360.146,A -85,B 0,C 180,E1 -1250.513,E2 -1250.513} C_VEL
LIN {X 0,Y 594.428,Z 369.889,A -85,B 0,C 180,E1 -1250.727,E2 -1250.727} C_VEL
LIN {X 0,Y 594.391,Z 381.491,A -85,B 0,C 180,E1 -1251.112,E2 -1251.112} C_VEL
LIN {X 0,Y 594.42,Z 391.42,A -85,B 0,C 180,E1 -1251.584,E2 -1251.584} C_VEL
LIN {X 0,Y 594.378,Z 401.111,A -85,B 0,C 180,E1 -1252.182,E2 -1252.182} C_VEL
LIN {X 0,Y 594.36,Z 408.862,A -85,B 0,C 180,E1 -1252.78,E2 -1252.78} C_VEL
LIN {X 0,Y 594.345,Z 416.749,A -85,B 0,C 180,E1 -1253.523,E2 -1253.523} C_VEL
LIN {X 0,Y 594.31,Z 424.108,A -85,B 0,C 180,E1 -1254.398,E2 -1254.398} C_VEL
LIN {X 0,Y 594.275,Z 429.731,A -85,B 0,C 180,E1 -1255.248,E2 -1255.248} C_VEL
LIN {X 0,Y 594.287,Z 434.953,A -85,B 0,C 180,E1 -1256.267,E2 -1256.267} C_VEL
LIN {X 0,Y 594.229,Z 438.78,A -85,B 0,C 180,E1 -1257.285,E2 -1257.285} C_VEL
LIN {X 0,Y 594.238,Z 440.579,A -85,B 0,C 180,E1 -1257.963,E2 -1257.963} C_VEL
LIN {X 0,Y 594.247,Z 441.884,A -85,B 0,C 180,E1 -1258.641,E2 -1258.641} C_VEL
LIN {X 0,Y 594.235,Z 442.703,A -85,B 0,C 180,E1 -1259.319,E2 -1259.319} C_VEL
LIN {X 0,Y 594.234,Z 442.995,A -85,B 0,C 180,E1 -1259.997,E2 -1259.997} C_VEL
LIN {X 0,Y 594.238,Z 442.748,A -85,B 0,C 180,E1 -1260.674,E2 -1260.674} C_VEL
LIN {X 0,Y 594.246,Z 442.018,A -85,B 0,C 180,E1 -1261.352,E2 -1261.352} C_VEL
LIN {X 0,Y 594.241,Z 440.808,A -85,B 0,C 180,E1 -1262.03,E2 -1262.03} C_VEL
LIN {X 0,Y 594.248,Z 437.964,A -85,B 0,C 180,E1 -1263.047,E2 -1263.047} C_VEL
LIN {X 0,Y 594.261,Z 433.869,A -85,B 0,C 180,E1 -1264.065,E2 -1264.065} C_VEL
LIN {X 0,Y 594.257,Z 428.286,A -85,B 0,C 180,E1 -1265.085,E2 -1265.085} C_VEL
LIN {X 0,Y 594.322,Z 422.213,A -85,B 0,C 180,E1 -1265.935,E2 -1265.935} C_VEL
LIN {X 0,Y 594.354,Z 414.554,A -85,B 0,C 180,E1 -1266.787,E2 -1266.787} C_VEL
LIN {X 0,Y 594.367,Z 405.952,A -85,B 0,C 180,E1 -1267.555,E2 -1267.555} C_VEL
LIN {X 0,Y 594.412,Z 396.094,A -85,B 0,C 180,E1 -1268.238,E2 -1268.238} C_VEL
LIN {X 0,Y 594.456,Z 386.465,A -85,B 0,C 180,E1 -1268.751,E2 -1268.751} C_VEL
LIN {X 0,Y 594.452,Z 378.274,A -85,B 0,C 180,E1 -1269.094,E2 -1269.094} C_VEL
LIN {X 0,Y 594.498,Z 368.658,A -85,B 0,C 180,E1 -1269.394,E2 -1269.394} C_VEL
LIN {X 0,Y 594.484,Z 359.515,A -85,B 0,C 180,E1 -1269.587,E2 -1269.587} C_VEL
LIN {X 0,Y 594.513,Z 341.784,A -85,B 0,C 180,E1 -1269.817,E2 -1269.817} C_VEL
LIN {X 0,Y 593.852,Z 335.972,A -85,B 0,C 180,E1 -1269.897,E2 -1269.897} C_VEL
LIN {X 0,Y 588.291,Z 317.225,A -85,B 0,C 180,E1 -1270.219,E2 -1270.219} C_VEL
LIN {X 0,Y 587.576,Z 311.415,A -85,B 0,C 180,E1 -1270.302,E2 -1270.302} C_VEL
LIN {X 0,Y 587.37,Z 285.878,A -85,B 0,C 180,E1 -1270.617,E2 -1270.617} C_VEL
LIN {X 0,Y 587.228,Z 284.645,A -85,B 0,C 180,E1 -1270.641,E2 -1270.641} C_VEL
LIN {X 0,Y 587.312,Z 271.06,A -85,B 0,C 180,E1 -1273.49,E2 -1273.49} C_VEL
LIN {X 0,Y 587.307,Z 257.691,A -85,B 0,C 180,E1 -1276.328,E2 -1276.328} C_VEL
LIN {X 0,Y 587.313,Z 252.136,A -85,B 0,C 180,E1 -1277.537,E2 -1277.537} C_VEL
LIN {X 0,Y 587.289,Z 252.137,A -85,B 0,C 180,E1 -1280.301,E2 -1280.301} C_VEL
LIN {X 0,Y 587.279,Z 252.145,A -85,B 0,C 180,E1 -1283.255,E2 -1283.255} C_VEL
LIN {X 0,Y 587.276,Z 252.137,A -85,B 0,C 180,E1 -1286.163,E2 -1286.163} C_VEL
LIN {X 0,Y 587.317,Z 252.142,A -85,B 0,C 180,E1 -1289.127,E2 -1289.127} C_VEL
LIN {X 0,Y 587.29,Z 252.139,A -85,B 0,C 180,E1 -1291.826,E2 -1291.826} C_VEL
LIN {X 0,Y 587.308,Z 252.133,A -85,B 0,C 180,E1 -1294.341,E2 -1294.341} C_VEL
LIN {X 0,Y 587.309,Z 252.142,A -85,B 0,C 180,E1 -1297.603,E2 -1297.603} C_VEL
LIN {X 0,Y 587.276,Z 252.139,A -85,B 0,C 180,E1 -1300.25,E2 -1300.25} C_VEL
LIN {X 0,Y 587.261,Z 252.142,A -85,B 0,C 180,E1 -1303.112,E2 -1303.112} C_VEL
LIN {X 0,Y 587.284,Z 252.142,A -85,B 0,C 180,E1 -1306.045,E2 -1306.045} C_VEL
LIN {X 0,Y 587.293,Z 252.136,A -85,B 0,C 180,E1 -1308.921,E2 -1308.921} C_VEL
LIN {X 0,Y 587.29,Z 252.141,A -85,B 0,C 180,E1 -1311.517,E2 -1311.517} C_VEL
LIN {X 0,Y 587.302,Z 252.142,A -85,B 0,C 180,E1 -1314.1,E2 -1314.1} C_VEL
LIN {X 0,Y 587.292,Z 252.136,A -85,B 0,C 180,E1 -1316.884,E2 -1316.884} C_VEL
LIN {X 0,Y 587.298,Z 252.141,A -85,B 0,C 180,E1 -1319.827,E2 -1319.827} C_VEL
LIN {X 0,Y 587.299,Z 252.143,A -85,B 0,C 180,E1 -1322.303,E2 -1322.303} C_VEL
LIN {X 0,Y 587.308,Z 252.14,A -85,B 0,C 180,E1 -1324.481,E2 -1324.481} C_VEL
LIN {X 0,Y 587.287,Z 252.137,A -85,B 0,C 180,E1 -1327.483,E2 -1327.483} C_VEL
LIN {X 0,Y 587.292,Z 252.146,A -85,B 0,C 180,E1 -1330.422,E2 -1330.422} C_VEL
LIN {X 0,Y 587.287,Z 252.136,A -85,B 0,C 180,E1 -1333.308,E2 -1333.308} C_VEL
LIN {X 0,Y 587.31,Z 252.138,A -85,B 0,C 180,E1 -1336.152,E2 -1336.152} C_VEL
LIN {X 0,Y 587.351,Z 252.133,A -85,B 0,C 180,E1 -1338.962,E2 -1338.962} C_VEL
LIN {X 0,Y 587.311,Z 252.133,A -85,B 0,C 180,E1 -1341.743,E2 -1341.743} C_VEL
LIN {X 0,Y 587.329,Z 252.138,A -85,B 0,C 180,E1 -1344.506,E2 -1344.506} C_VEL
LIN {X 0,Y 587.326,Z 252.135,A -85,B 0,C 180,E1 -1347.255,E2 -1347.255} C_VEL
LIN {X 0,Y 587.312,Z 252.133,A -85,B 0,C 180,E1 -1349.999,E2 -1349.999} C_VEL
LIN {X 0,Y 587.331,Z 252.138,A -85,B 0,C 180,E1 -1352.742,E2 -1352.742} C_VEL
LIN {X 0,Y 587.321,Z 252.135,A -85,B 0,C 180,E1 -1355.492,E2 -1355.492} C_VEL
LIN {X 0,Y 587.31,Z 252.133,A -85,B 0,C 180,E1 -1358.255,E2 -1358.255} C_VEL
LIN {X 0,Y 587.345,Z 252.139,A -85,B 0,C 180,E1 -1361.166,E2 -1361.166} C_VEL
LIN {X 0,Y 587.3,Z 252.134,A -85,B 0,C 180,E1 -1364.262,E2 -1364.262} C_VEL
LIN {X 0,Y 587.313,Z 252.143,A -85,B 0,C 180,E1 -1367.406,E2 -1367.406} C_VEL
LIN {X 0,Y 587.273,Z 252.138,A -85,B 0,C 180,E1 -1370.305,E2 -1370.305} C_VEL
LIN {X 0,Y 587.261,Z 252.141,A -85,B 0,C 180,E1 -1372.872,E2 -1372.872} C_VEL
LIN {X 0,Y 587.305,Z 252.144,A -85,B 0,C 180,E1 -1375.516,E2 -1375.516} C_VEL
LIN {X 0,Y 587.288,Z 252.144,A -85,B 0,C 180,E1 -1377.819,E2 -1377.819} C_VEL
LIN {X 0,Y 587.292,Z 252.136,A -85,B 0,C 180,E1 -1380.515,E2 -1380.515} C_VEL
LIN {X 0,Y 587.287,Z 252.14,A -85,B 0,C 180,E1 -1383.398,E2 -1383.398} C_VEL
LIN {X 0,Y 587.303,Z 252.145,A -85,B 0,C 180,E1 -1385.897,E2 -1385.897} C_VEL
LIN {X 0,Y 587.286,Z 252.139,A -85,B 0,C 180,E1 -1388.481,E2 -1388.481} C_VEL
LIN {X 0,Y 587.31,Z 252.134,A -85,B 0,C 180,E1 -1391.157,E2 -1391.157} C_VEL
LIN {X 0,Y 587.284,Z 252.147,A -85,B 0,C 180,E1 -1394.117,E2 -1394.117} C_VEL
LIN {X 0,Y 587.268,Z 252.139,A -85,B 0,C 180,E1 -1396.997,E2 -1396.997} C_VEL
LIN {X 0,Y 587.272,Z 252.141,A -85,B 0,C 180,E1 -1399.749,E2 -1399.749} C_VEL
LIN {X 0,Y 587.301,Z 252.144,A -85,B 0,C 180,E1 -1402.396,E2 -1402.396} C_VEL
LIN {X 0,Y 587.306,Z 252.136,A -85,B 0,C 180,E1 -1404.949,E2 -1404.949} C_VEL
LIN {X 0,Y 587.293,Z 252.135,A -85,B 0,C 180,E1 -1407.424,E2 -1407.424} C_VEL
LIN {X 0,Y 587.278,Z 252.139,A -85,B 0,C 180,E1 -1409.833,E2 -1409.833} C_VEL
LIN {X 0,Y 587.31,Z 252.14,A -85,B 0,C 180,E1 -1412.311,E2 -1412.311} C_VEL
LIN {X 0,Y 587.299,Z 252.143,A -85,B 0,C 180,E1 -1414.487,E2 -1414.487} C_VEL
LIN {X 0,Y 587.302,Z 252.135,A -85,B 0,C 180,E1 -1417.49,E2 -1417.49} C_VEL
LIN {X 0,Y 587.279,Z 252.142,A -85,B 0,C 180,E1 -1420.428,E2 -1420.428} C_VEL
LIN {X 0,Y 587.31,Z 252.137,A -85,B 0,C 180,E1 -1423.315,E2 -1423.315} C_VEL
LIN {X 0,Y 587.31,Z 252.134,A -85,B 0,C 180,E1 -1426.157,E2 -1426.157} C_VEL
LIN {X 0,Y 587.325,Z 252.142,A -85,B 0,C 180,E1 -1428.966,E2 -1428.966} C_VEL
LIN {X 0,Y 587.3,Z 252.136,A -85,B 0,C 180,E1 -1431.748,E2 -1431.748} C_VEL
LIN {X 0,Y 587.278,Z 252.139,A -85,B 0,C 180,E1 -1433.821,E2 -1433.821} C_VEL
LIN {X 0,Y 587.269,Z 252.14,A -85,B 0,C 180,E1 -1435.886,E2 -1435.886} C_VEL
LIN {X 0,Y 587.325,Z 252.133,A -85,B 0,C 180,E1 -1437.946,E2 -1437.946} C_VEL
LIN {X 0,Y 587.342,Z 252.13,A -85,B 0,C 180,E1 -1440.003,E2 -1440.003} C_VEL
LIN {X 0,Y 587.33,Z 252.132,A -85,B 0,C 180,E1 -1442.747,E2 -1442.747} C_VEL
LIN {X 0,Y 587.335,Z 252.141,A -85,B 0,C 180,E1 -1445.496,E2 -1445.496} C_VEL
LIN {X 0,Y 587.318,Z 252.133,A -85,B 0,C 180,E1 -1448.259,E2 -1448.259} C_VEL
LIN {X 0,Y 587.317,Z 252.135,A -85,B 0,C 180,E1 -1451.127,E2 -1451.127} C_VEL
LIN {X 0,Y 587.315,Z 252.135,A -85,B 0,C 180,E1 -1454.249,E2 -1454.249} C_VEL
LIN {X 0,Y 587.272,Z 252.138,A -85,B 0,C 180,E1 -1456.796,E2 -1456.796} C_VEL
LIN {X 0,Y 587.291,Z 252.142,A -85,B 0,C 180,E1 -1459.579,E2 -1459.579} C_VEL
LIN {X 0,Y 587.295,Z 252.144,A -85,B 0,C 180,E1 -1461.778,E2 -1461.778} C_VEL
LIN {X 0,Y 587.298,Z 252.135,A -85,B 0,C 180,E1 -1464.763,E2 -1464.763} C_VEL
LIN {X 0,Y 587.292,Z 252.14,A -85,B 0,C 180,E1 -1467.686,E2 -1467.686} C_VEL
LIN {X 0,Y 587.321,Z 252.142,A -85,B 0,C 180,E1 -1470.173,E2 -1470.173} C_VEL
LIN {X 0,Y 587.326,Z 252.131,A -85,B 0,C 180,E1 -1473.113,E2 -1473.113} C_VEL
LIN {X 0,Y 587.268,Z 252.143,A -85,B 0,C 180,E1 -1475.904,E2 -1475.904} C_VEL
LIN {X 0,Y 587.303,Z 252.143,A -85,B 0,C 180,E1 -1478.483,E2 -1478.483} C_VEL
LIN {X 0,Y 587.296,Z 252.136,A -85,B 0,C 180,E1 -1481.162,E2 -1481.162} C_VEL
LIN {X 0,Y 587.295,Z 252.139,A -85,B 0,C 180,E1 -1484.113,E2 -1484.113} C_VEL
LIN {X 0,Y 587.284,Z 252.141,A -85,B 0,C 180,E1 -1486.993,E2 -1486.993} C_VEL
LIN {X 0,Y 587.288,Z 252.136,A -85,B 0,C 180,E1 -1489.746,E2 -1489.746} C_VEL
LIN {X 0,Y 587.332,Z 252.136,A -85,B 0,C 180,E1 -1492.393,E2 -1492.393} C_VEL
LIN {X 0,Y 587.324,Z 252.132,A -85,B 0,C 180,E1 -1495.657,E2 -1495.657} C_VEL
LIN {X 0,Y 587.311,Z 252.134,A -85,B 0,C 180,E1 -1498.231,E2 -1498.231} C_VEL
LIN {X 0,Y 587.339,Z 252.139,A -85,B 0,C 180,E1 -1500.87,E2 -1500.87} C_VEL
LIN {X 0,Y 587.292,Z 252.136,A -85,B 0,C 180,E1 -1503.834,E2 -1503.834} C_VEL
LIN {X 0,Y 587.298,Z 252.14,A -85,B 0,C 180,E1 -1506.742,E2 -1506.742} C_VEL
LIN {X 0,Y 587.325,Z 252.211,A -85,B 0,C 180,E1 -1508.089,E2 -1508.089} C_VEL
LIN {X 0,Y 587.631,Z 258.631,A -85,B 0,C 180,E1 -1509.159,E2 -1509.159} C_VEL
LIN {X 0,Y 587.538,Z 275.379,A -85,B 0,C 180,E1 -1511.882,E2 -1511.882} C_VEL
LIN {X 0,Y 587.39,Z 291.011,A -85,B 0,C 180,E1 -1514.384,E2 -1514.384} C_VEL
LIN {X 0,Y 587.369,Z 308.876,A -85,B 0,C 180,E1 -1517.213,E2 -1517.213} C_VEL
LIN {X 0,Y 587.299,Z 322.763,A -85,B 0,C 180,E1 -1519.388,E2 -1519.388} C_VEL
LIN {X 0,Y 587.606,Z 328.986,A -85,B 0,C 180,E1 -1519.47,E2 -1519.47} C_VEL
LIN {X 0,Y 587.535,Z 399.218,A -85,B 0,C 180,E1 -1520.339,E2 -1520.339} C_VEL
LIN {X 0,Y 587.465,Z 408.464,A -85,B 0,C 180,E1 -1520.533,E2 -1520.533} C_VEL
LIN {X 0,Y 587.433,Z 416.928,A -85,B 0,C 180,E1 -1520.793,E2 -1520.793} C_VEL
LIN {X 0,Y 587.39,Z 425.427,A -85,B 0,C 180,E1 -1521.14,E2 -1521.14} C_VEL
LIN {X 0,Y 587.392,Z 433.75,A -85,B 0,C 180,E1 -1521.573,E2 -1521.573} C_VEL
LIN {X 0,Y 587.33,Z 441.784,A -85,B 0,C 180,E1 -1522.092,E2 -1522.092} C_VEL
LIN {X 0,Y 587.288,Z 449.431,A -85,B 0,C 180,E1 -1522.696,E2 -1522.696} C_VEL
LIN {X 0,Y 587.282,Z 457.823,A -85,B 0,C 180,E1 -1523.514,E2 -1523.514} C_VEL
LIN {X 0,Y 587.238,Z 464.441,A -85,B 0,C 180,E1 -1524.335,E2 -1524.335} C_VEL
LIN {X 0,Y 587.17,Z 469.994,A -85,B 0,C 180,E1 -1525.195,E2 -1525.195} C_VEL
LIN {X 0,Y 587.21,Z 475.153,A -85,B 0,C 180,E1 -1526.227,E2 -1526.227} C_VEL
LIN {X 0,Y 587.155,Z 477.792,A -85,B 0,C 180,E1 -1526.914,E2 -1526.914} C_VEL
LIN {X 0,Y 587.141,Z 480.683,A -85,B 0,C 180,E1 -1527.943,E2 -1527.943} C_VEL
LIN {X 0,Y 587.145,Z 481.938,A -85,B 0,C 180,E1 -1528.629,E2 -1528.629} C_VEL
LIN {X 0,Y 587.136,Z 482.712,A -85,B 0,C 180,E1 -1529.315,E2 -1529.315} C_VEL
LIN {X 0,Y 587.134,Z 483,A -85,B 0,C 180,E1 -1530.001,E2 -1530.001} C_VEL
LIN {X 0,Y 587.136,Z 482.711,A -85,B 0,C 180,E1 -1530.687,E2 -1530.687} C_VEL
LIN {X 0,Y 587.145,Z 481.934,A -85,B 0,C 180,E1 -1531.373,E2 -1531.373} C_VEL
LIN {X 0,Y 587.141,Z 480.677,A -85,B 0,C 180,E1 -1532.059,E2 -1532.059} C_VEL
LIN {X 0,Y 587.156,Z 477.784,A -85,B 0,C 180,E1 -1533.089,E2 -1533.089} C_VEL
LIN {X 0,Y 587.211,Z 475.142,A -85,B 0,C 180,E1 -1533.775,E2 -1533.775} C_VEL
LIN {X 0,Y 587.17,Z 469.979,A -85,B 0,C 180,E1 -1534.807,E2 -1534.807} C_VEL
LIN {X 0,Y 587.253,Z 463.179,A -85,B 0,C 180,E1 -1535.84,E2 -1535.84} C_VEL
LIN {X 0,Y 587.271,Z 456.289,A -85,B 0,C 180,E1 -1536.645,E2 -1536.645} C_VEL
LIN {X 0,Y 587.29,Z 449.406,A -85,B 0,C 180,E1 -1537.306,E2 -1537.306} C_VEL
LIN {X 0,Y 587.331,Z 441.753,A -85,B 0,C 180,E1 -1537.911,E2 -1537.911} C_VEL
LIN {X 0,Y 587.393,Z 433.711,A -85,B 0,C 180,E1 -1538.429,E2 -1538.429} C_VEL
LIN {X 0,Y 587.391,Z 425.377,A -85,B 0,C 180,E1 -1538.863,E2 -1538.863} C_VEL
LIN {X 0,Y 587.434,Z 416.865,A -85,B 0,C 180,E1 -1539.209,E2 -1539.209} C_VEL
LIN {X 0,Y 587.461,Z 406.713,A -85,B 0,C 180,E1 -1539.512,E2 -1539.512} C_VEL
LIN {X 0,Y 587.544,Z 394.973,A -85,B 0,C 180,E1 -1539.728,E2 -1539.728} C_VEL
LIN {X 0,Y 587.424,Z 323.873,A -85,B 0,C 180,E1 -1540.595,E2 -1540.595} C_VEL
LIN {X 0,Y 587.26,Z 322.539,A -85,B 0,C 180,E1 -1540.647,E2 -1540.647} C_VEL
LIN {X 0,Y 587.359,Z 305.511,A -85,B 0,C 180,E1 -1543.318,E2 -1543.318} C_VEL
LIN {X 0,Y 587.468,Z 286.53,A -85,B 0,C 180,E1 -1546.329,E2 -1546.329} C_VEL
LIN {X 0,Y 587.583,Z 268.208,A -85,B 0,C 180,E1 -1549.279,E2 -1549.279} C_VEL
LIN {X 0,Y 587.582,Z 254.151,A -85,B 0,C 180,E1 -1551.581,E2 -1551.581} C_VEL
LIN {X 0,Y 587.298,Z 252.14,A -85,B 0,C 180,E1 -1551.961,E2 -1551.961} C_VEL
LIN {X 0,Y 587.287,Z 252.146,A -85,B 0,C 180,E1 -1554.762,E2 -1554.762} C_VEL
LIN {X 0,Y 587.293,Z 252.137,A -85,B 0,C 180,E1 -1557.681,E2 -1557.681} C_VEL
LIN {X 0,Y 587.27,Z 252.143,A -85,B 0,C 180,E1 -1560.497,E2 -1560.497} C_VEL
LIN {X 0,Y 587.273,Z 252.145,A -85,B 0,C 180,E1 -1563.101,E2 -1563.101} C_VEL
LIN {X 0,Y 587.259,Z 252.14,A -85,B 0,C 180,E1 -1565.903,E2 -1565.903} C_VEL
LIN {X 0,Y 587.296,Z 252.138,A -85,B 0,C 180,E1 -1568.483,E2 -1568.483} C_VEL
LIN {X 0,Y 587.306,Z 252.141,A -85,B 0,C 180,E1 -1571.16,E2 -1571.16} C_VEL
LIN {X 0,Y 587.297,Z 252.135,A -85,B 0,C 180,E1 -1574.109,E2 -1574.109} C_VEL
LIN {X 0,Y 587.296,Z 252.146,A -85,B 0,C 180,E1 -1576.99,E2 -1576.99} C_VEL
LIN {X 0,Y 587.309,Z 252.134,A -85,B 0,C 180,E1 -1579.743,E2 -1579.743} C_VEL
LIN {X 0,Y 587.322,Z 252.133,A -85,B 0,C 180,E1 -1582.389,E2 -1582.389} C_VEL
LIN {X 0,Y 587.345,Z 252.131,A -85,B 0,C 180,E1 -1585.654,E2 -1585.654} C_VEL
LIN {X 0,Y 587.344,Z 252.13,A -85,B 0,C 180,E1 -1588.229,E2 -1588.229} C_VEL
LIN {X 0,Y 587.354,Z 252.135,A -85,B 0,C 180,E1 -1590.867,E2 -1590.867} C_VEL
LIN {X 0,Y 587.316,Z 252.134,A -85,B 0,C 180,E1 -1593.829,E2 -1593.829} C_VEL
LIN {X 0,Y 587.326,Z 252.132,A -85,B 0,C 180,E1 -1595.991,E2 -1595.991} C_VEL
LIN {X 0,Y 587.324,Z 252.132,A -85,B 0,C 180,E1 -1598.223,E2 -1598.223} C_VEL
LIN {X 0,Y 587.352,Z 252.139,A -85,B 0,C 180,E1 -1601.149,E2 -1601.149} C_VEL
LIN {X 0,Y 587.359,Z 252.225,A -85,B 0,C 180,E1 -1602.592,E2 -1602.592} C_VEL
LIN {X 0,Y 587.304,Z 263.918,A -85,B 0,C 180,E1 -1605.089,E2 -1605.089} C_VEL
LIN {X 0,Y 587.262,Z 275.611,A -85,B 0,C 180,E1 -1607.557,E2 -1607.557} C_VEL
LIN {X 0,Y 587.172,Z 284.649,A -85,B 0,C 180,E1 -1609.449,E2 -1609.449} C_VEL
LIN {X 0,Y 587.574,Z 289.223,A -85,B 0,C 180,E1 -1609.518,E2 -1609.518} C_VEL
LIN {X 0,Y 587.486,Z 360.179,A -85,B 0,C 180,E1 -1610.399,E2 -1610.399} C_VEL
LIN {X 0,Y 587.436,Z 369.914,A -85,B 0,C 180,E1 -1610.616,E2 -1610.616} C_VEL
LIN {X 0,Y 587.391,Z 381.503,A -85,B 0,C 180,E1 -1611.005,E2 -1611.005} C_VEL
LIN {X 0,Y 587.389,Z 392.95,A -85,B 0,C 180,E1 -1611.569,E2 -1611.569} C_VEL
LIN {X 0,Y 587.353,Z 402.35,A -85,B 0,C 180,E1 -1612.174,E2 -1612.174} C_VEL
LIN {X 0,Y 587.302,Z 411.845,A -85,B 0,C 180,E1 -1612.951,E2 -1612.951} C_VEL
LIN {X 0,Y 587.268,Z 419.997,A -85,B 0,C 180,E1 -1613.814,E2 -1613.814} C_VEL
LIN {X 0,Y 587.196,Z 426.478,A -85,B 0,C 180,E1 -1614.675,E2 -1614.675} C_VEL
LIN {X 0,Y 587.199,Z 431.656,A -85,B 0,C 180,E1 -1615.535,E2 -1615.535} C_VEL
LIN {X 0,Y 587.193,Z 436.42,A -85,B 0,C 180,E1 -1616.566,E2 -1616.566} C_VEL
LIN {X 0,Y 587.136,Z 438.782,A -85,B 0,C 180,E1 -1617.252,E2 -1617.252} C_VEL
LIN {X 0,Y 587.137,Z 440.587,A -85,B 0,C 180,E1 -1617.939,E2 -1617.939} C_VEL
LIN {X 0,Y 587.147,Z 441.893,A -85,B 0,C 180,E1 -1618.625,E2 -1618.625} C_VEL
LIN {X 0,Y 587.136,Z 442.707,A -85,B 0,C 180,E1 -1619.311,E2 -1619.311} C_VEL
LIN {X 0,Y 587.135,Z 442.995,A -85,B 0,C 180,E1 -1619.997,E2 -1619.997} C_VEL
LIN {X 0,Y 587.139,Z 442.753,A -85,B 0,C 180,E1 -1620.682,E2 -1620.682} C_VEL
LIN {X 0,Y 587.146,Z 442.025,A -85,B 0,C 180,E1 -1621.368,E2 -1621.368} C_VEL
LIN {X 0,Y 587.14,Z 440.813,A -85,B 0,C 180,E1 -1622.054,E2 -1622.054} C_VEL
LIN {X 0,Y 587.157,Z 437.968,A -85,B 0,C 180,E1 -1623.084,E2 -1623.084} C_VEL
LIN {X 0,Y 587.181,Z 433.876,A -85,B 0,C 180,E1 -1624.115,E2 -1624.115} C_VEL
LIN {X 0,Y 587.171,Z 428.283,A -85,B 0,C 180,E1 -1625.147,E2 -1625.147} C_VEL
LIN {X 0,Y 587.263,Z 422.216,A -85,B 0,C 180,E1 -1626.007,E2 -1626.007} C_VEL
LIN {X 0,Y 587.281,Z 414.557,A -85,B 0,C 180,E1 -1626.869,E2 -1626.869} C_VEL
LIN {X 0,Y 587.32,Z 405.949,A -85,B 0,C 180,E1 -1627.646,E2 -1627.646} C_VEL
LIN {X 0,Y 587.396,Z 396.1,A -85,B 0,C 180,E1 -1628.337,E2 -1628.337} C_VEL
LIN {X 0,Y 587.422,Z 386.46,A -85,B 0,C 180,E1 -1628.857,E2 -1628.857} C_VEL
LIN {X 0,Y 587.445,Z 377.06,A -85,B 0,C 180,E1 -1629.247,E2 -1629.247} C_VEL
LIN {X 0,Y 587.49,Z 366.972,A -85,B 0,C 180,E1 -1629.55,E2 -1629.55} C_VEL
LIN {X 0,Y 587.543,Z 355.502,A -85,B 0,C 180,E1 -1629.767,E2 -1629.767} C_VEL
LIN {X 0,Y 587.576,Z 311.415,A -85,B 0,C 180,E1 -1630.302,E2 -1630.302} C_VEL
LIN {X 0,Y 586.85,Z 307.534,A -85,B 0,C 180,E1 -1630.362,E2 -1630.362} C_VEL
LIN {X 0,Y 581.203,Z 295.529,A -85,B 0,C 180,E1 -1630.612,E2 -1630.612} C_VEL
LIN {X 0,Y 580.588,Z 291.648,A -85,B 0,C 180,E1 -1630.671,E2 -1630.671} C_VEL
LIN {X 0,Y 580.337,Z 285.906,A -85,B 0,C 180,E1 -1630.746,E2 -1630.746} C_VEL
LIN {X 0,Y 580.173,Z 284.637,A -85,B 0,C 180,E1 -1630.773,E2 -1630.773} C_VEL
LIN {X 0,Y 580.225,Z 271.057,A -85,B 0,C 180,E1 -1633.658,E2 -1633.658} C_VEL
LIN {X 0,Y 580.274,Z 257.688,A -85,B 0,C 180,E1 -1636.532,E2 -1636.532} C_VEL
LIN {X 0,Y 580.274,Z 253.013,A -85,B 0,C 180,E1 -1637.57,E2 -1637.57} C_VEL
LIN {X 0,Y 580.256,Z 253.013,A -85,B 0,C 180,E1 -1639.819,E2 -1639.819} C_VEL
LIN {X 0,Y 580.228,Z 253.016,A -85,B 0,C 180,E1 -1642.049,E2 -1642.049} C_VEL
LIN {X 0,Y 580.255,Z 253.022,A -85,B 0,C 180,E1 -1645.077,E2 -1645.077} C_VEL
LIN {X 0,Y 580.223,Z 253.018,A -85,B 0,C 180,E1 -1647.844,E2 -1647.844} C_VEL
LIN {X 0,Y 580.237,Z 253.016,A -85,B 0,C 180,E1 -1650.686,E2 -1650.686} C_VEL
LIN {X 0,Y 580.275,Z 253.02,A -85,B 0,C 180,E1 -1653.311,E2 -1653.311} C_VEL
LIN {X 0,Y 580.212,Z 253.023,A -85,B 0,C 180,E1 -1655.751,E2 -1655.751} C_VEL
LIN {X 0,Y 580.25,Z 253.014,A -85,B 0,C 180,E1 -1658.142,E2 -1658.142} C_VEL
LIN {X 0,Y 580.262,Z 253.012,A -85,B 0,C 180,E1 -1660.839,E2 -1660.839} C_VEL
LIN {X 0,Y 580.232,Z 253.025,A -85,B 0,C 180,E1 -1663.654,E2 -1663.654} C_VEL
LIN {X 0,Y 580.238,Z 253.015,A -85,B 0,C 180,E1 -1666.605,E2 -1666.605} C_VEL
LIN {X 0,Y 580.258,Z 253.013,A -85,B 0,C 180,E1 -1669.152,E2 -1669.152} C_VEL
LIN {X 0,Y 580.251,Z 253.023,A -85,B 0,C 180,E1 -1671.922,E2 -1671.922} C_VEL
LIN {X 0,Y 580.239,Z 253.017,A -85,B 0,C 180,E1 -1674.451,E2 -1674.451} C_VEL
LIN {X 0,Y 580.243,Z 253.014,A -85,B 0,C 180,E1 -1676.971,E2 -1676.971} C_VEL
LIN {X 0,Y 580.253,Z 253.014,A -85,B 0,C 180,E1 -1679.422,E2 -1679.422} C_VEL
LIN {X 0,Y 580.247,Z 253.023,A -85,B 0,C 180,E1 -1682.137,E2 -1682.137} C_VEL
LIN {X 0,Y 580.265,Z 253.012,A -85,B 0,C 180,E1 -1684.917,E2 -1684.917} C_VEL
LIN {X 0,Y 580.222,Z 253.021,A -85,B 0,C 180,E1 -1687.944,E2 -1687.944} C_VEL
LIN {X 0,Y 580.261,Z 253.014,A -85,B 0,C 180,E1 -1690.911,E2 -1690.911} C_VEL
LIN {X 0,Y 580.226,Z 253.017,A -85,B 0,C 180,E1 -1693.823,E2 -1693.823} C_VEL
LIN {X 0,Y 580.229,Z 253.024,A -85,B 0,C 180,E1 -1696.694,E2 -1696.694} C_VEL
LIN {X 0,Y 580.259,Z 253.012,A -85,B 0,C 180,E1 -1699.531,E2 -1699.531} C_VEL
LIN {X 0,Y 580.284,Z 253.014,A -85,B 0,C 180,E1 -1702.343,E2 -1702.343} C_VEL
LIN {X 0,Y 580.288,Z 253.013,A -85,B 0,C 180,E1 -1705.136,E2 -1705.136} C_VEL
LIN {X 0,Y 580.27,Z 253.01,A -85,B 0,C 180,E1 -1707.917,E2 -1707.917} C_VEL
LIN {X 0,Y 580.322,Z 253.011,A -85,B 0,C 180,E1 -1710.693,E2 -1710.693} C_VEL
LIN {X 0,Y 580.251,Z 253.016,A -85,B 0,C 180,E1 -1713.471,E2 -1713.471} C_VEL
LIN {X 0,Y 580.282,Z 253.012,A -85,B 0,C 180,E1 -1715.559,E2 -1715.559} C_VEL
LIN {X 0,Y 580.275,Z 253.01,A -85,B 0,C 180,E1 -1718.356,E2 -1718.356} C_VEL
LIN {X 0,Y 580.317,Z 253.015,A -85,B 0,C 180,E1 -1721.233,E2 -1721.233} C_VEL
LIN {X 0,Y 580.251,Z 253.013,A -85,B 0,C 180,E1 -1724.34,E2 -1724.34} C_VEL
LIN {X 0,Y 580.25,Z 253.017,A -85,B 0,C 180,E1 -1726.916,E2 -1726.916} C_VEL
LIN {X 0,Y 580.249,Z 253.017,A -85,B 0,C 180,E1 -1729.823,E2 -1729.823} C_VEL
LIN {X 0,Y 580.227,Z 253.018,A -85,B 0,C 180,E1 -1732.053,E2 -1732.053} C_VEL
LIN {X 0,Y 580.26,Z 253.015,A -85,B 0,C 180,E1 -1735.08,E2 -1735.08} C_VEL
LIN {X 0,Y 580.259,Z 253.019,A -85,B 0,C 180,E1 -1737.865,E2 -1737.865} C_VEL
LIN {X 0,Y 580.241,Z 253.014,A -85,B 0,C 180,E1 -1740.699,E2 -1740.699} C_VEL
LIN {X 0,Y 580.252,Z 253.016,A -85,B 0,C 180,E1 -1743.32,E2 -1743.32} C_VEL
LIN {X 0,Y 580.272,Z 253.02,A -85,B 0,C 180,E1 -1745.77,E2 -1745.77} C_VEL
LIN {X 0,Y 580.239,Z 253.021,A -85,B 0,C 180,E1 -1748.148,E2 -1748.148} C_VEL
LIN {X 0,Y 580.274,Z 253.01,A -85,B 0,C 180,E1 -1750.843,E2 -1750.843} C_VEL
LIN {X 0,Y 580.239,Z 253.018,A -85,B 0,C 180,E1 -1753.659,E2 -1753.659} C_VEL
LIN {X 0,Y 580.233,Z 253.018,A -85,B 0,C 180,E1 -1756.611,E2 -1756.611} C_VEL
LIN {X 0,Y 580.252,Z 253.013,A -85,B 0,C 180,E1 -1759.16,E2 -1759.16} C_VEL
LIN {X 0,Y 580.244,Z 253.018,A -85,B 0,C 180,E1 -1761.93,E2 -1761.93} C_VEL
LIN {X 0,Y 580.265,Z 253.02,A -85,B 0,C 180,E1 -1764.46,E2 -1764.46} C_VEL
LIN {X 0,Y 580.251,Z 253.015,A -85,B 0,C 180,E1 -1766.979,E2 -1766.979} C_VEL
LIN {X 0,Y 580.248,Z 253.013,A -85,B 0,C 180,E1 -1769.428,E2 -1769.428} C_VEL
LIN {X 0,Y 580.255,Z 253.016,A -85,B 0,C 180,E1 -1772.145,E2 -1772.145} C_VEL
LIN {X 0,Y 580.254,Z 253.018,A -85,B 0,C 180,E1 -1774.923,E2 -1774.923} C_VEL
LIN {X 0,Y 580.233,Z 253.016,A -85,B 0,C 180,E1 -1777.951,E2 -1777.951} C_VEL
LIN {X 0,Y 580.267,Z 253.02,A -85,B 0,C 180,E1 -1780.917,E2 -1780.917} C_VEL
LIN {X 0,Y 580.239,Z 253.014,A -85,B 0,C 180,E1 -1783.829,E2 -1783.829} C_VEL
LIN {X 0,Y 580.238,Z 253.021,A -85,B 0,C 180,E1 -1786.699,E2 -1786.699} C_VEL
LIN {X 0,Y 580.307,Z 253.013,A -85,B 0,C 180,E1 -1788.831,E2 -1788.831} C_VEL
LIN {X 0,Y 580.276,Z 253.012,A -85,B 0,C 180,E1 -1791.647,E2 -1791.647} C_VEL
LIN {X 0,Y 580.239,Z 253.016,A -85,B 0,C 180,E1 -1793.746,E2 -1793.746} C_VEL
LIN {X 0,Y 580.227,Z 253.017,A -85,B 0,C 180,E1 -1795.836,E2 -1795.836} C_VEL
LIN {X 0,Y 580.298,Z 253.008,A -85,B 0,C 180,E1 -1797.921,E2 -1797.921} C_VEL
LIN {X 0,Y 580.313,Z 253.006,A -85,B 0,C 180,E1 -1800.003,E2 -1800.003} C_VEL
LIN {X 0,Y 580.3,Z 253.008,A -85,B 0,C 180,E1 -1802.78,E2 -1802.78} C_VEL
LIN {X 0,Y 580.3,Z 253.016,A -85,B 0,C 180,E1 -1805.563,E2 -1805.563} C_VEL
LIN {X 0,Y 580.287,Z 253.009,A -85,B 0,C 180,E1 -1808.36,E2 -1808.36} C_VEL
LIN {X 0,Y 580.288,Z 253.012,A -85,B 0,C 180,E1 -1811.194,E2 -1811.194} C_VEL
LIN {X 0,Y 580.291,Z 253.013,A -85,B 0,C 180,E1 -1814.021,E2 -1814.021} C_VEL
LIN {X 0,Y 580.238,Z 253.015,A -85,B 0,C 180,E1 -1816.902,E2 -1816.902} C_VEL
LIN {X 0,Y 580.266,Z 253.021,A -85,B 0,C 180,E1 -1819.826,E2 -1819.826} C_VEL
LIN {X 0,Y 580.266,Z 253.011,A -85,B 0,C 180,E1 -1822.806,E2 -1822.806} C_VEL
LIN {X 0,Y 580.266,Z 253.011,A -85,B 0,C 180,E1 -1825.084,E2 -1825.084} C_VEL
LIN {X 0,Y 580.268,Z 253.02,A -85,B 0,C 180,E1 -1828.189,E2 -1828.189} C_VEL
LIN {X 0,Y 580.27,Z 253.013,A -85,B 0,C 180,E1 -1830.696,E2 -1830.696} C_VEL
LIN {X 0,Y 580.271,Z 253.01,A -85,B 0,C 180,E1 -1833.315,E2 -1833.315} C_VEL
LIN {X 0,Y 580.217,Z 253.02,A -85,B 0,C 180,E1 -1835.755,E2 -1835.755} C_VEL
LIN {X 0,Y 580.269,Z 253.018,A -85,B 0,C 180,E1 -1838.15,E2 -1838.15} C_VEL
LIN {X 0,Y 580.267,Z 253.015,A -85,B 0,C 180,E1 -1840.848,E2 -1840.848} C_VEL
LIN {X 0,Y 580.232,Z 253.015,A -85,B 0,C 180,E1 -1843.664,E2 -1843.664} C_VEL
LIN {X 0,Y 580.234,Z 253.025,A -85,B 0,C 180,E1 -1846.615,E2 -1846.615} C_VEL
LIN {X 0,Y 580.284,Z 253.011,A -85,B 0,C 180,E1 -1849.158,E2 -1849.158} C_VEL
LIN {X 0,Y 580.276,Z 253.01,A -85,B 0,C 180,E1 -1851.93,E2 -1851.93} C_VEL
LIN {X 0,Y 580.219,Z 253.022,A -85,B 0,C 180,E1 -1854.452,E2 -1854.452} C_VEL
LIN {X 0,Y 580.278,Z 253.018,A -85,B 0,C 180,E1 -1856.976,E2 -1856.976} C_VEL
LIN {X 0,Y 580.265,Z 253.014,A -85,B 0,C 180,E1 -1859.425,E2 -1859.425} C_VEL
LIN {X 0,Y 580.242,Z 253.014,A -85,B 0,C 180,E1 -1862.153,E2 -1862.153} C_VEL
LIN {X 0,Y 580.239,Z 253.023,A -85,B 0,C 180,E1 -1864.919,E2 -1864.919} C_VEL
LIN {X 0,Y 580.281,Z 253.02,A -85,B 0,C 180,E1 -1867.199,E2 -1867.199} C_VEL
LIN {X 0,Y 580.277,Z 253.132,A -85,B 0,C 180,E1 -1867.973,E2 -1867.973} C_VEL
LIN {X 0,Y 580.702,Z 258.325,A -85,B 0,C 180,E1 -1868.847,E2 -1868.847} C_VEL
LIN {X 0,Y 580.551,Z 276.496,A -85,B 0,C 180,E1 -1871.838,E2 -1871.838} C_VEL
LIN {X 0,Y 580.37,Z 293.244,A -85,B 0,C 180,E1 -1874.551,E2 -1874.551} C_VEL
LIN {X 0,Y 580.292,Z 311.109,A -85,B 0,C 180,E1 -1877.41,E2 -1877.41} C_VEL
LIN {X 0,Y 580.214,Z 322.754,A -85,B 0,C 180,E1 -1879.256,E2 -1879.256} C_VEL
LIN {X 0,Y 580.643,Z 329.027,A -85,B 0,C 180,E1 -1879.343,E2 -1879.343} C_VEL
LIN {X 0,Y 580.556,Z 399.218,A -85,B 0,C 180,E1 -1880.222,E2 -1880.222} C_VEL
LIN {X 0,Y 580.476,Z 408.464,A -85,B 0,C 180,E1 -1880.418,E2 -1880.418} C_VEL
LIN {X 0,Y 580.441,Z 416.928,A -85,B 0,C 180,E1 -1880.682,E2 -1880.682} C_VEL
LIN {X 0,Y 580.378,Z 425.428,A -85,B 0,C 180,E1 -1881.032,E2 -1881.032} C_VEL
LIN {X 0,Y 580.364,Z 433.754,A -85,B 0,C 180,E1 -1881.47,E2 -1881.47} C_VEL
LIN {X 0,Y 580.284,Z 441.786,A -85,B 0,C 180,E1 -1881.995,E2 -1881.995} C_VEL
LIN {X 0,Y 580.223,Z 450.445,A -85,B 0,C 180,E1 -1882.695,E2 -1882.695} C_VEL
LIN {X 0,Y 580.204,Z 459.013,A -85,B 0,C 180,E1 -1883.576,E2 -1883.576} C_VEL
LIN {X 0,Y 580.151,Z 465.619,A -85,B 0,C 180,E1 -1884.44,E2 -1884.44} C_VEL
LIN {X 0,Y 580.084,Z 469.994,A -85,B 0,C 180,E1 -1885.136,E2 -1885.136} C_VEL
LIN {X 0,Y 580.122,Z 475.153,A -85,B 0,C 180,E1 -1886.181,E2 -1886.181} C_VEL
LIN {X 0,Y 580.07,Z 477.793,A -85,B 0,C 180,E1 -1886.876,E2 -1886.876} C_VEL
LIN {X 0,Y 580.04,Z 480.684,A -85,B 0,C 180,E1 -1887.918,E2 -1887.918} C_VEL
LIN {X 0,Y 580.045,Z 481.938,A -85,B 0,C 180,E1 -1888.613,E2 -1888.613} C_VEL
LIN {X 0,Y 580.036,Z 482.711,A -85,B 0,C 180,E1 -1889.307,E2 -1889.307} C_VEL
LIN {X 0,Y 580.034,Z 483,A -85,B 0,C 180,E1 -1890.001,E2 -1890.001} C_VEL
LIN {X 0,Y 580.036,Z 482.71,A -85,B 0,C 180,E1 -1890.695,E2 -1890.695} C_VEL
LIN {X 0,Y 580.045,Z 481.934,A -85,B 0,C 180,E1 -1891.39,E2 -1891.39} C_VEL
LIN {X 0,Y 580.04,Z 480.678,A -85,B 0,C 180,E1 -1892.084,E2 -1892.084} C_VEL
LIN {X 0,Y 580.071,Z 477.784,A -85,B 0,C 180,E1 -1893.126,E2 -1893.126} C_VEL
LIN {X 0,Y 580.123,Z 475.143,A -85,B 0,C 180,E1 -1893.822,E2 -1893.822} C_VEL
LIN {X 0,Y 580.084,Z 469.979,A -85,B 0,C 180,E1 -1894.866,E2 -1894.866} C_VEL
LIN {X 0,Y 580.194,Z 463.178,A -85,B 0,C 180,E1 -1895.911,E2 -1895.911} C_VEL
LIN {X 0,Y 580.228,Z 455.494,A -85,B 0,C 180,E1 -1896.808,E2 -1896.808} C_VEL
LIN {X 0,Y 580.252,Z 448.394,A -85,B 0,C 180,E1 -1897.482,E2 -1897.482} C_VEL
LIN {X 0,Y 580.304,Z 440.531,A -85,B 0,C 180,E1 -1898.095,E2 -1898.095} C_VEL
LIN {X 0,Y 580.386,Z 430.714,A -85,B 0,C 180,E1 -1898.707,E2 -1898.707} C_VEL
LIN {X 0,Y 580.417,Z 419.273,A -85,B 0,C 180,E1 -1899.233,E2 -1899.233} C_VEL
LIN {X 0,Y 580.475,Z 409.206,A -85,B 0,C 180,E1 -1899.562,E2 -1899.562} C_VEL
LIN {X 0,Y 580.547,Z 400.381,A -85,B 0,C 180,E1 -1899.759,E2 -1899.759} C_VEL
LIN {X 0,Y 580.484,Z 324.746,A -85,B 0,C 180,E1 -1900.713,E2 -1900.713} C_VEL
LIN {X 0,Y 580.208,Z 322.732,A -85,B 0,C 180,E1 -1900.748,E2 -1900.748} C_VEL
LIN {X 0,Y 580.305,Z 305.511,A -85,B 0,C 180,E1 -1903.483,E2 -1903.483} C_VEL
LIN {X 0,Y 580.463,Z 287.646,A -85,B 0,C 180,E1 -1906.351,E2 -1906.351} C_VEL
LIN {X 0,Y 580.608,Z 269.922,A -85,B 0,C 180,E1 -1909.237,E2 -1909.237} C_VEL
LIN {X 0,Y 580.587,Z 255.201,A -85,B 0,C 180,E1 -1911.667,E2 -1911.667} C_VEL
LIN {X 0,Y 580.251,Z 253.018,A -85,B 0,C 180,E1 -1912.054,E2 -1912.054} C_VEL
LIN {X 0,Y 580.242,Z 253.023,A -85,B 0,C 180,E1 -1914.712,E2 -1914.712} C_VEL
LIN {X 0,Y 580.242,Z 253.017,A -85,B 0,C 180,E1 -1917.405,E2 -1917.405} C_VEL
LIN {X 0,Y 580.231,Z 253.016,A -85,B 0,C 180,E1 -1919.777,E2 -1919.777} C_VEL
LIN {X 0,Y 580.246,Z 253.015,A -85,B 0,C 180,E1 -1922.205,E2 -1922.205} C_VEL
LIN {X 0,Y 580.224,Z 253.024,A -85,B 0,C 180,E1 -1924.702,E2 -1924.702} C_VEL
LIN {X 0,Y 580.271,Z 253.015,A -85,B 0,C 180,E1 -1927.271,E2 -1927.271} C_VEL
LIN {X 0,Y 580.278,Z 253.01,A -85,B 0,C 180,E1 -1930.267,E2 -1930.267} C_VEL
LIN {X 0,Y 580.255,Z 253.018,A -85,B 0,C 180,E1 -1932.709,E2 -1932.709} C_VEL
LIN {X 0,Y 580.258,Z 253.013,A -85,B 0,C 180,E1 -1935.611,E2 -1935.611} C_VEL
LIN {X 0,Y 580.248,Z 253.013,A -85,B 0,C 180,E1 -1938.227,E2 -1938.227} C_VEL
LIN {X 0,Y 580.272,Z 253.02,A -85,B 0,C 180,E1 -1940.963,E2 -1940.963} C_VEL
LIN {X 0,Y 580.254,Z 253.014,A -85,B 0,C 180,E1 -1943.593,E2 -1943.593} C_VEL
LIN {X 0,Y 580.286,Z 253.009,A -85,B 0,C 180,E1 -1946.141,E2 -1946.141} C_VEL
LIN {X 0,Y 580.278,Z 253.013,A -85,B 0,C 180,E1 -1948.613,E2 -1948.613} C_VEL
LIN {X 0,Y 580.297,Z 253.017,A -85,B 0,C 180,E1 -1951.022,E2 -1951.022} C_VEL
LIN {X 0,Y 580.264,Z 253.012,A -85,B 0,C 180,E1 -1954.147,E2 -1954.147} C_VEL
LIN {X 0,Y 580.276,Z 253.012,A -85,B 0,C 180,E1 -1956.44,E2 -1956.44} C_VEL
LIN {X 0,Y 580.281,Z 253.015,A -85,B 0,C 180,E1 -1959.435,E2 -1959.435} C_VEL
LIN {X 0,Y 580.266,Z 253.015,A -85,B 0,C 180,E1 -1961.642,E2 -1961.642} C_VEL
LIN {X 0,Y 580.328,Z 253.146,A -85,B 0,C 180,E1 -1962.574,E2 -1962.574} C_VEL
LIN {X 0,Y 580.27,Z 265.591,A -85,B 0,C 180,E1 -1965.263,E2 -1965.263} C_VEL
LIN {X 0,Y 580.193,Z 278.955,A -85,B 0,C 180,E1 -1968.113,E2 -1968.113} C_VEL
LIN {X 0,Y 580.115,Z 284.617,A -85,B 0,C 180,E1 -1969.311,E2 -1969.311} C_VEL
LIN {X 0,Y 580.594,Z 289.435,A -85,B 0,C 180,E1 -1969.392,E2 -1969.392} C_VEL
LIN {X 0,Y 580.513,Z 360.213,A -85,B 0,C 180,E1 -1970.283,E2 -1970.283} C_VEL
LIN {X 0,Y 580.444,Z 369.938,A -85,B 0,C 180,E1 -1970.501,E2 -1970.501} C_VEL
LIN {X 0,Y 580.392,Z 381.514,A -85,B 0,C 180,E1 -1970.896,E2 -1970.896} C_VEL
LIN {X 0,Y 580.346,Z 392.975,A -85,B 0,C 180,E1 -1971.466,E2 -1971.466} C_VEL
LIN {X 0,Y 580.303,Z 402.372,A -85,B 0,C 180,E1 -1972.079,E2 -1972.079} C_VEL
LIN {X 0,Y 580.251,Z 411.85,A -85,B 0,C 180,E1 -1972.865,E2 -1972.865} C_VEL
LIN {X 0,Y 580.195,Z 420.012,A -85,B 0,C 180,E1 -1973.738,E2 -1973.738} C_VEL
LIN {X 0,Y 580.122,Z 426.489,A -85,B 0,C 180,E1 -1974.609,E2 -1974.609} C_VEL
LIN {X 0,Y 580.123,Z 431.666,A -85,B 0,C 180,E1 -1975.48,E2 -1975.48} C_VEL
LIN {X 0,Y 580.123,Z 436.417,A -85,B 0,C 180,E1 -1976.524,E2 -1976.524} C_VEL
LIN {X 0,Y 580.047,Z 438.785,A -85,B 0,C 180,E1 -1977.219,E2 -1977.219} C_VEL
LIN {X 0,Y 580.037,Z 440.595,A -85,B 0,C 180,E1 -1977.914,E2 -1977.914} C_VEL
LIN {X 0,Y 580.047,Z 441.901,A -85,B 0,C 180,E1 -1978.608,E2 -1978.608} C_VEL
LIN {X 0,Y 580.036,Z 442.71,A -85,B 0,C 180,E1 -1979.302,E2 -1979.302} C_VEL
LIN {X 0,Y 580.036,Z 442.995,A -85,B 0,C 180,E1 -1979.997,E2 -1979.997} C_VEL
LIN {X 0,Y 580.039,Z 442.758,A -85,B 0,C 180,E1 -1980.691,E2 -1980.691} C_VEL
LIN {X 0,Y 580.046,Z 442.033,A -85,B 0,C 180,E1 -1981.385,E2 -1981.385} C_VEL
LIN {X 0,Y 580.04,Z 440.819,A -85,B 0,C 180,E1 -1982.08,E2 -1982.08} C_VEL
LIN {X 0,Y 580.072,Z 437.973,A -85,B 0,C 180,E1 -1983.122,E2 -1983.122} C_VEL
LIN {X 0,Y 580.106,Z 433.88,A -85,B 0,C 180,E1 -1984.165,E2 -1984.165} C_VEL
LIN {X 0,Y 580.091,Z 428.279,A -85,B 0,C 180,E1 -1985.21,E2 -1985.21} C_VEL
LIN {X 0,Y 580.207,Z 422.211,A -85,B 0,C 180,E1 -1986.08,E2 -1986.08} C_VEL
LIN {X 0,Y 580.222,Z 414.561,A -85,B 0,C 180,E1 -1986.953,E2 -1986.953} C_VEL
LIN {X 0,Y 580.274,Z 405.945,A -85,B 0,C 180,E1 -1987.74,E2 -1987.74} C_VEL
LIN {X 0,Y 580.375,Z 396.101,A -85,B 0,C 180,E1 -1988.439,E2 -1988.439} C_VEL
LIN {X 0,Y 580.41,Z 386.456,A -85,B 0,C 180,E1 -1988.965,E2 -1988.965} C_VEL
LIN {X 0,Y 580.451,Z 377.048,A -85,B 0,C 180,E1 -1989.36,E2 -1989.36} C_VEL
LIN {X 0,Y 580.474,Z 366.948,A -85,B 0,C 180,E1 -1989.667,E2 -1989.667} C_VEL
LIN {X 0,Y 580.563,Z 355.461,A -85,B 0,C 180,E1 -1989.885,E2 -1989.885} C_VEL
LIN {X 0,Y 580.588,Z 291.648,A -85,B 0,C 180,E1 -1990.671,E2 -1990.671} C_VEL
LIN {X 0,Y 580.243,Z 288.216,A -85,B 0,C 180,E1 -1990.787,E2 -1990.787} C_VEL
LIN {X 0,Y 579.353,Z 285.344,A -85,B 0,C 180,E1 -1991.001,E2 -1991.001} C_VEL
LIN {X 0,Y 578.154,Z 282.968,A -85,B 0,C 180,E1 -1991.281,E2 -1991.281} C_VEL
LIN {X 0,Y 576.171,Z 280.281,A -85,B 0,C 180,E1 -1991.778,E2 -1991.778} C_VEL
LIN {X 0,Y 574.292,Z 277.785,A -85,B 0,C 180,E1 -1992.352,E2 -1992.352} C_VEL
LIN {X 0,Y 573.225,Z 275.151,A -85,B 0,C 180,E1 -1992.944,E2 -1992.944} C_VEL
LIN {X 0,Y 573.15,Z 274.231,A -85,B 0,C 180,E1 -1993.143,E2 -1993.143} C_VEL
LIN {X 0,Y 573.216,Z 261.028,A -85,B 0,C 180,E1 -1996.009,E2 -1996.009} C_VEL
LIN {X 0,Y 573.235,Z 253.89,A -85,B 0,C 180,E1 -1997.591,E2 -1997.591} C_VEL
LIN {X 0,Y 573.213,Z 253.89,A -85,B 0,C 180,E1 -2000.073,E2 -2000.073} C_VEL
LIN {X 0,Y 573.199,Z 253.892,A -85,B 0,C 180,E1 -2002.334,E2 -2002.334} C_VEL
LIN {X 0,Y 573.203,Z 253.897,A -85,B 0,C 180,E1 -2005.407,E2 -2005.407} C_VEL
LIN {X 0,Y 573.179,Z 253.894,A -85,B 0,C 180,E1 -2008.014,E2 -2008.014} C_VEL
LIN {X 0,Y 573.196,Z 253.892,A -85,B 0,C 180,E1 -2010.173,E2 -2010.173} C_VEL
LIN {X 0,Y 573.221,Z 253.89,A -85,B 0,C 180,E1 -2012.641,E2 -2012.641} C_VEL
LIN {X 0,Y 573.175,Z 253.901,A -85,B 0,C 180,E1 -2015.184,E2 -2015.184} C_VEL
LIN {X 0,Y 573.197,Z 253.897,A -85,B 0,C 180,E1 -2017.804,E2 -2017.804} C_VEL
LIN {X 0,Y 573.213,Z 253.89,A -85,B 0,C 180,E1 -2020.52,E2 -2020.52} C_VEL
LIN {X 0,Y 573.198,Z 253.901,A -85,B 0,C 180,E1 -2023.663,E2 -2023.663} C_VEL
LIN {X 0,Y 573.2,Z 253.891,A -85,B 0,C 180,E1 -2026.636,E2 -2026.636} C_VEL
LIN {X 0,Y 573.219,Z 253.894,A -85,B 0,C 180,E1 -2029.472,E2 -2029.472} C_VEL
LIN {X 0,Y 573.195,Z 253.897,A -85,B 0,C 180,E1 -2032.188,E2 -2032.188} C_VEL
LIN {X 0,Y 573.207,Z 253.891,A -85,B 0,C 180,E1 -2034.811,E2 -2034.811} C_VEL
LIN {X 0,Y 573.206,Z 253.892,A -85,B 0,C 180,E1 -2037.351,E2 -2037.351} C_VEL
LIN {X 0,Y 573.202,Z 253.895,A -85,B 0,C 180,E1 -2040.507,E2 -2040.507} C_VEL
LIN {X 0,Y 573.223,Z 253.89,A -85,B 0,C 180,E1 -2043.496,E2 -2043.496} C_VEL
LIN {X 0,Y 573.179,Z 253.903,A -85,B 0,C 180,E1 -2046.131,E2 -2046.131} C_VEL
LIN {X 0,Y 573.195,Z 253.896,A -85,B 0,C 180,E1 -2048.706,E2 -2048.706} C_VEL
LIN {X 0,Y 573.182,Z 253.894,A -85,B 0,C 180,E1 -2051.409,E2 -2051.409} C_VEL
LIN {X 0,Y 573.196,Z 253.892,A -85,B 0,C 180,E1 -2053.619,E2 -2053.619} C_VEL
LIN {X 0,Y 573.187,Z 253.903,A -85,B 0,C 180,E1 -2056.527,E2 -2056.527} C_VEL
LIN {X 0,Y 573.229,Z 253.888,A -85,B 0,C 180,E1 -2059.402,E2 -2059.402} C_VEL
LIN {X 0,Y 573.233,Z 253.891,A -85,B 0,C 180,E1 -2062.248,E2 -2062.248} C_VEL
LIN {X 0,Y 573.261,Z 253.889,A -85,B 0,C 180,E1 -2065.076,E2 -2065.076} C_VEL
LIN {X 0,Y 573.242,Z 253.886,A -85,B 0,C 180,E1 -2067.891,E2 -2067.891} C_VEL
LIN {X 0,Y 573.29,Z 253.887,A -85,B 0,C 180,E1 -2070.701,E2 -2070.701} C_VEL
LIN {X 0,Y 573.2,Z 253.894,A -85,B 0,C 180,E1 -2073.513,E2 -2073.513} C_VEL
LIN {X 0,Y 573.245,Z 253.888,A -85,B 0,C 180,E1 -2075.627,E2 -2075.627} C_VEL
LIN {X 0,Y 573.248,Z 253.887,A -85,B 0,C 180,E1 -2078.459,E2 -2078.459} C_VEL
LIN {X 0,Y 573.261,Z 253.893,A -85,B 0,C 180,E1 -2081.311,E2 -2081.311} C_VEL
LIN {X 0,Y 573.217,Z 253.889,A -85,B 0,C 180,E1 -2084.426,E2 -2084.426} C_VEL
LIN {X 0,Y 573.198,Z 253.898,A -85,B 0,C 180,E1 -2087.112,E2 -2087.112} C_VEL
LIN {X 0,Y 573.199,Z 253.893,A -85,B 0,C 180,E1 -2090.077,E2 -2090.077} C_VEL
LIN {X 0,Y 573.185,Z 253.893,A -85,B 0,C 180,E1 -2092.338,E2 -2092.338} C_VEL
LIN {X 0,Y 573.21,Z 253.898,A -85,B 0,C 180,E1 -2095.41,E2 -2095.41} C_VEL
LIN {X 0,Y 573.203,Z 253.895,A -85,B 0,C 180,E1 -2098.033,E2 -2098.033} C_VEL
LIN {X 0,Y 573.186,Z 253.893,A -85,B 0,C 180,E1 -2100.887,E2 -2100.887} C_VEL
LIN {X 0,Y 573.229,Z 253.894,A -85,B 0,C 180,E1 -2103.53,E2 -2103.53} C_VEL
LIN {X 0,Y 573.205,Z 253.898,A -85,B 0,C 180,E1 -2106.05,E2 -2106.05} C_VEL
LIN {X 0,Y 573.199,Z 253.892,A -85,B 0,C 180,E1 -2108.703,E2 -2108.703} C_VEL
LIN {X 0,Y 573.207,Z 253.893,A -85,B 0,C 180,E1 -2111.457,E2 -2111.457} C_VEL
LIN {X 0,Y 573.188,Z 253.899,A -85,B 0,C 180,E1 -2114.336,E2 -2114.336} C_VEL
LIN {X 0,Y 573.191,Z 253.893,A -85,B 0,C 180,E1 -2117.361,E2 -2117.361} C_VEL
LIN {X 0,Y 573.203,Z 253.899,A -85,B 0,C 180,E1 -2120.397,E2 -2120.397} C_VEL
LIN {X 0,Y 573.21,Z 253.891,A -85,B 0,C 180,E1 -2123.081,E2 -2123.081} C_VEL
LIN {X 0,Y 573.231,Z 253.888,A -85,B 0,C 180,E1 -2125.675,E2 -2125.675} C_VEL
LIN {X 0,Y 573.205,Z 253.897,A -85,B 0,C 180,E1 -2128.189,E2 -2128.189} C_VEL
LIN {X 0,Y 573.22,Z 253.898,A -85,B 0,C 180,E1 -2130.638,E2 -2130.638} C_VEL
LIN {X 0,Y 573.201,Z 253.891,A -85,B 0,C 180,E1 -2133.51,E2 -2133.51} C_VEL
LIN {X 0,Y 573.181,Z 253.896,A -85,B 0,C 180,E1 -2136.138,E2 -2136.138} C_VEL
LIN {X 0,Y 573.217,Z 253.899,A -85,B 0,C 180,E1 -2138.713,E2 -2138.713} C_VEL
LIN {X 0,Y 573.183,Z 253.895,A -85,B 0,C 180,E1 -2141.415,E2 -2141.415} C_VEL
LIN {X 0,Y 573.212,Z 253.89,A -85,B 0,C 180,E1 -2143.625,E2 -2143.625} C_VEL
LIN {X 0,Y 573.193,Z 253.896,A -85,B 0,C 180,E1 -2146.533,E2 -2146.533} C_VEL
LIN {X 0,Y 573.258,Z 253.89,A -85,B 0,C 180,E1 -2148.738,E2 -2148.738} C_VEL
LIN {X 0,Y 573.223,Z 253.892,A -85,B 0,C 180,E1 -2151.544,E2 -2151.544} C_VEL
LIN {X 0,Y 573.203,Z 253.894,A -85,B 0,C 180,E1 -2153.669,E2 -2153.669} C_VEL
LIN {X 0,Y 573.186,Z 253.895,A -85,B 0,C 180,E1 -2155.785,E2 -2155.785} C_VEL
LIN {X 0,Y 573.272,Z 253.884,A -85,B 0,C 180,E1 -2157.896,E2 -2157.896} C_VEL
LIN {X 0,Y 573.283,Z 253.882,A -85,B 0,C 180,E1 -2160.004,E2 -2160.004} C_VEL
LIN {X 0,Y 573.269,Z 253.885,A -85,B 0,C 180,E1 -2162.814,E2 -2162.814} C_VEL
LIN {X 0,Y 573.265,Z 253.891,A -85,B 0,C 180,E1 -2165.632,E2 -2165.632} C_VEL
LIN {X 0,Y 573.23,Z 253.888,A -85,B 0,C 180,E1 -2168.463,E2 -2168.463} C_VEL
LIN {X 0,Y 573.259,Z 253.889,A -85,B 0,C 180,E1 -2171.315,E2 -2171.315} C_VEL
LIN {X 0,Y 573.251,Z 253.886,A -85,B 0,C 180,E1 -2174.42,E2 -2174.42} C_VEL
LIN {X 0,Y 573.183,Z 253.895,A -85,B 0,C 180,E1 -2177.117,E2 -2177.117} C_VEL
LIN {X 0,Y 573.255,Z 253.887,A -85,B 0,C 180,E1 -2179.333,E2 -2179.333} C_VEL
LIN {X 0,Y 573.207,Z 253.894,A -85,B 0,C 180,E1 -2182.341,E2 -2182.341} C_VEL
LIN {X 0,Y 573.213,Z 253.89,A -85,B 0,C 180,E1 -2184.871,E2 -2184.871} C_VEL
LIN {X 0,Y 573.224,Z 253.894,A -85,B 0,C 180,E1 -2187.771,E2 -2187.771} C_VEL
LIN {X 0,Y 573.23,Z 253.897,A -85,B 0,C 180,E1 -2190.179,E2 -2190.179} C_VEL
LIN {X 0,Y 573.244,Z 253.889,A -85,B 0,C 180,E1 -2192.648,E2 -2192.648} C_VEL
LIN {X 0,Y 573.178,Z 253.894,A -85,B 0,C 180,E1 -2195.192,E2 -2195.192} C_VEL
LIN {X 0,Y 573.209,Z 253.893,A -85,B 0,C 180,E1 -2197.812,E2 -2197.812} C_VEL
LIN {X 0,Y 573.24,Z 253.895,A -85,B 0,C 180,E1 -2200.527,E2 -2200.527} C_VEL
LIN {X 0,Y 573.2,Z 253.892,A -85,B 0,C 180,E1 -2203.365,E2 -2203.365} C_VEL
LIN {X 0,Y 573.203,Z 253.898,A -85,B 0,C 180,E1 -2206.337,E2 -2206.337} C_VEL
LIN {X 0,Y 573.242,Z 253.886,A -85,B 0,C 180,E1 -2209.477,E2 -2209.477} C_VEL
LIN {X 0,Y 573.221,Z 253.891,A -85,B 0,C 180,E1 -2212.193,E2 -2212.193} C_VEL
LIN {X 0,Y 573.217,Z 253.893,A -85,B 0,C 180,E1 -2215.233,E2 -2215.233} C_VEL
LIN {X 0,Y 573.233,Z 253.887,A -85,B 0,C 180,E1 -2217.776,E2 -2217.776} C_VEL
LIN {X 0,Y 573.231,Z 253.893,A -85,B 0,C 180,E1 -2220.634,E2 -2220.634} C_VEL
LIN {X 0,Y 573.196,Z 253.895,A -85,B 0,C 180,E1 -2223.517,E2 -2223.517} C_VEL
LIN {X 0,Y 573.199,Z 253.893,A -85,B 0,C 180,E1 -2226.135,E2 -2226.135} C_VEL
LIN {X 0,Y 573.225,Z 253.985,A -85,B 0,C 180,E1 -2227.853,E2 -2227.853} C_VEL
LIN {X 0,Y 573.716,Z 258.29,A -85,B 0,C 180,E1 -2228.592,E2 -2228.592} C_VEL
LIN {X 0,Y 573.58,Z 275.379,A -85,B 0,C 180,E1 -2231.425,E2 -2231.425} C_VEL
LIN {X 0,Y 573.383,Z 292.128,A -85,B 0,C 180,E1 -2234.175,E2 -2234.175} C_VEL
LIN {X 0,Y 573.295,Z 309.993,A -85,B 0,C 180,E1 -2237.073,E2 -2237.073} C_VEL
LIN {X 0,Y 573.171,Z 322.872,A -85,B 0,C 180,E1 -2239.125,E2 -2239.125} C_VEL
LIN {X 0,Y 573.654,Z 328.425,A -85,B 0,C 180,E1 -2239.204,E2 -2239.204} C_VEL
LIN {X 0,Y 573.582,Z 399.218,A -85,B 0,C 180,E1 -2240.102,E2 -2240.102} C_VEL
LIN {X 0,Y 573.495,Z 408.463,A -85,B 0,C 180,E1 -2240.301,E2 -2240.301} C_VEL
LIN {X 0,Y 573.425,Z 418.134,A -85,B 0,C 180,E1 -2240.611,E2 -2240.611} C_VEL
LIN {X 0,Y 573.345,Z 427.288,A -85,B 0,C 180,E1 -2241.01,E2 -2241.01} C_VEL
LIN {X 0,Y 573.299,Z 438.095,A -85,B 0,C 180,E1 -2241.631,E2 -2241.631} C_VEL
LIN {X 0,Y 573.206,Z 447.396,A -85,B 0,C 180,E1 -2242.339,E2 -2242.339} C_VEL
LIN {X 0,Y 573.164,Z 454.053,A -85,B 0,C 180,E1 -2242.958,E2 -2242.958} C_VEL
LIN {X 0,Y 573.129,Z 460.37,A -85,B 0,C 180,E1 -2243.665,E2 -2243.665} C_VEL
LIN {X 0,Y 573.086,Z 465.62,A -85,B 0,C 180,E1 -2244.371,E2 -2244.371} C_VEL
LIN {X 0,Y 572.995,Z 469.995,A -85,B 0,C 180,E1 -2245.076,E2 -2245.076} C_VEL
LIN {X 0,Y 573.024,Z 475.154,A -85,B 0,C 180,E1 -2246.133,E2 -2246.133} C_VEL
LIN {X 0,Y 572.991,Z 477.792,A -85,B 0,C 180,E1 -2246.837,E2 -2246.837} C_VEL
LIN {X 0,Y 572.94,Z 480.685,A -85,B 0,C 180,E1 -2247.892,E2 -2247.892} C_VEL
LIN {X 0,Y 572.944,Z 481.936,A -85,B 0,C 180,E1 -2248.595,E2 -2248.595} C_VEL
LIN {X 0,Y 572.937,Z 482.71,A -85,B 0,C 180,E1 -2249.298,E2 -2249.298} C_VEL
